// Mitsubishi GX Works2 project: OLD CRF BUFFER 22-01-223_F1   PLC: Q02/Q02H

PROGRAM MAIN
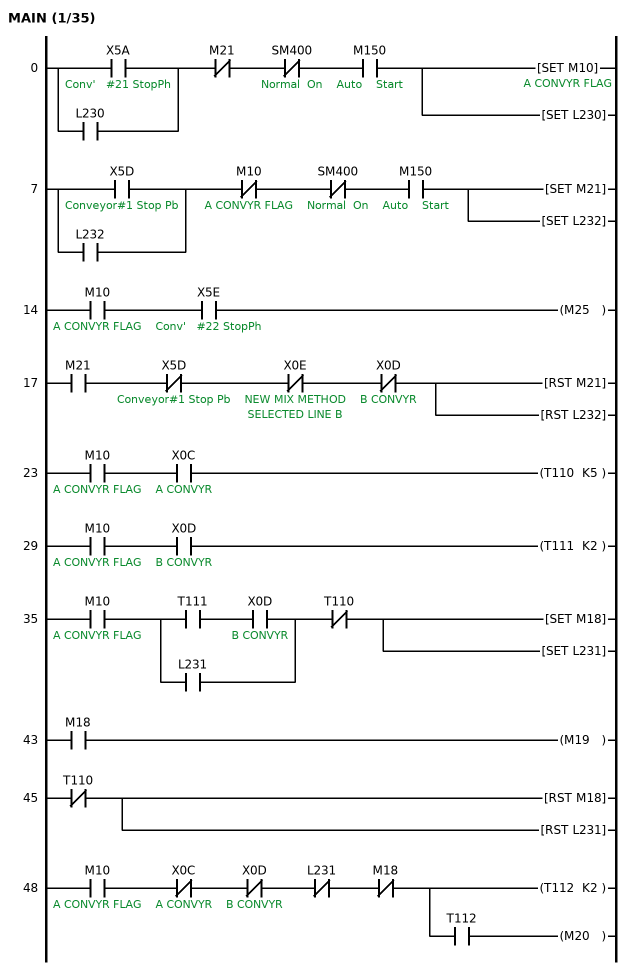
0     LD      X5A  ; Conv'   #21 StopPh
      OR      L230
      ANI     M21
      ANI     SM400  ; Normal  On
      AND     M150  ; Auto    Start
      SET     M10  ; A CONVYR FLAG
      SET     L230
7     LD      X5D  ; Conveyor#1 Stop Pb
      OR      L232
      ANI     M10  ; A CONVYR FLAG
      ANI     SM400  ; Normal  On
      AND     M150  ; Auto    Start
      SET     M21
      SET     L232
14    LD      M10  ; A CONVYR FLAG
      AND     X5E  ; Conv'   #22 StopPh
      OUT     M25
17    LD      M21
      ANI     X5D  ; Conveyor#1 Stop Pb
      ANI     X0E  ; NEW MIX METHOD  SELECTED LINE B
      ANI     X0D  ; B CONVYR
      RST     M21
      RST     L232
23    LD      M10  ; A CONVYR FLAG
      AND     X0C  ; A CONVYR
      OUT     T110 K5
29    LD      M10  ; A CONVYR FLAG
      AND     X0D  ; B CONVYR
      OUT     T111 K2
35    LD      M10  ; A CONVYR FLAG
      LD      T111
      AND     X0D  ; B CONVYR
      OR      L231
      ANB
      ANI     T110
      SET     M18
      SET     L231
43    LD      M18
      OUT     M19
45    LDI     T110
      RST     M18
      RST     L231
48    LD      M10  ; A CONVYR FLAG
      ANI     X0C  ; A CONVYR
      ANI     X0D  ; B CONVYR
      ANI     L231
      ANI     M18
      OUT     T112 K2
      AND     T112
      OUT     M20
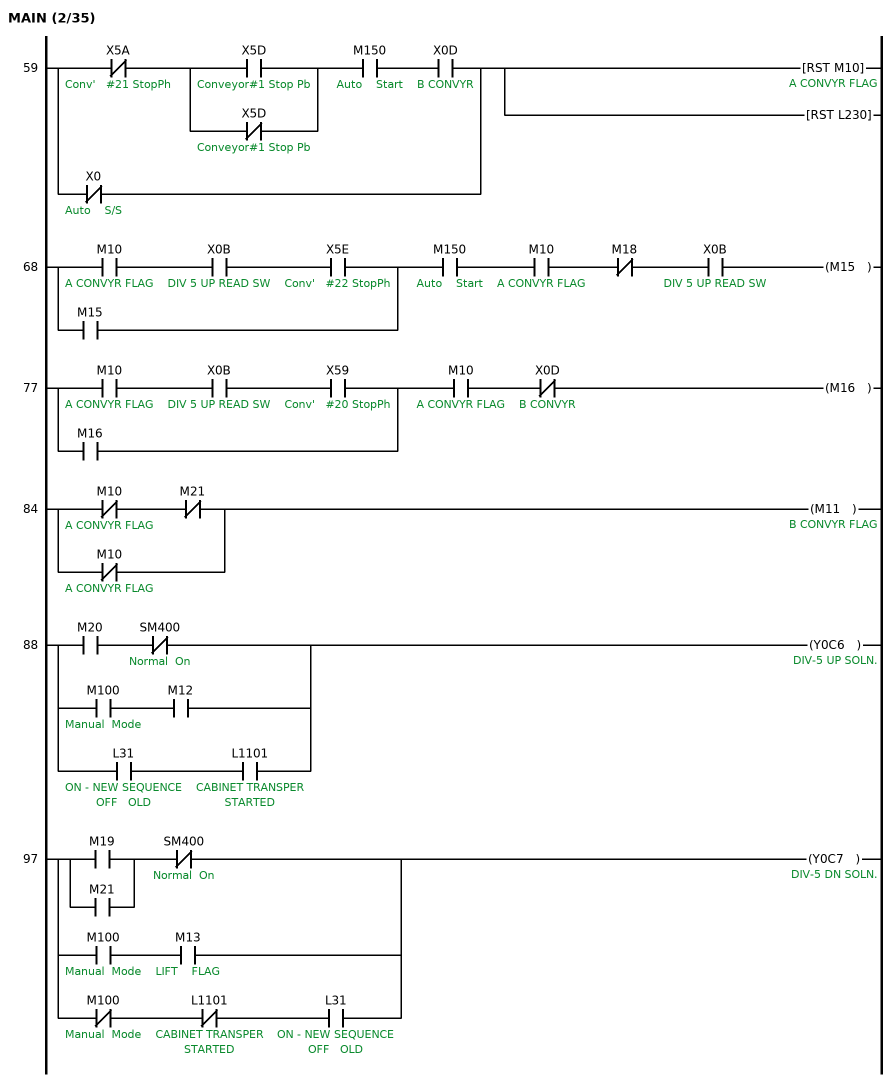
59    LDI     X5A  ; Conv'   #21 StopPh
      LD      X5D  ; Conveyor#1 Stop Pb
      ORI     X5D  ; Conveyor#1 Stop Pb
      ANB
      AND     M150  ; Auto    Start
      AND     X0D  ; B CONVYR
      ORI     X0  ; Auto    S/S
      RST     M10  ; A CONVYR FLAG
      RST     L230
68    LD      M10  ; A CONVYR FLAG
      AND     X0B  ; DIV 5 UP READ SW
      AND     X5E  ; Conv'   #22 StopPh
      OR      M15
      AND     M150  ; Auto    Start
      AND     M10  ; A CONVYR FLAG
      ANI     M18
      AND     X0B  ; DIV 5 UP READ SW
      OUT     M15
77    LD      M10  ; A CONVYR FLAG
      AND     X0B  ; DIV 5 UP READ SW
      AND     X59  ; Conv'   #20 StopPh
      OR      M16
      AND     M10  ; A CONVYR FLAG
      ANI     X0D  ; B CONVYR
      OUT     M16
84    LDI     M10  ; A CONVYR FLAG
      ANI     M21
      ORI     M10  ; A CONVYR FLAG
      OUT     M11  ; B CONVYR FLAG
88    LD      M20
      ANI     SM400  ; Normal  On
      LD      M100  ; Manual  Mode
      AND     M12
      ORB
      LD      L31  ; ON - NEW SEQUENCE OFF   OLD
      AND     L1101  ; CABINET TRANSPER STARTED
      ORB
      OUT     Y0C6  ; DIV-5 UP SOLN.
97    LD      M19
      OR      M21
      ANI     SM400  ; Normal  On
      LD      M100  ; Manual  Mode
      AND     M13  ; LIFT    FLAG
      ORB
      LDI     M100  ; Manual  Mode
      ANI     L1101  ; CABINET TRANSPER STARTED
      AND     L31  ; ON - NEW SEQUENCE OFF   OLD
      ORB
      OUT     Y0C7  ; DIV-5 DN SOLN.
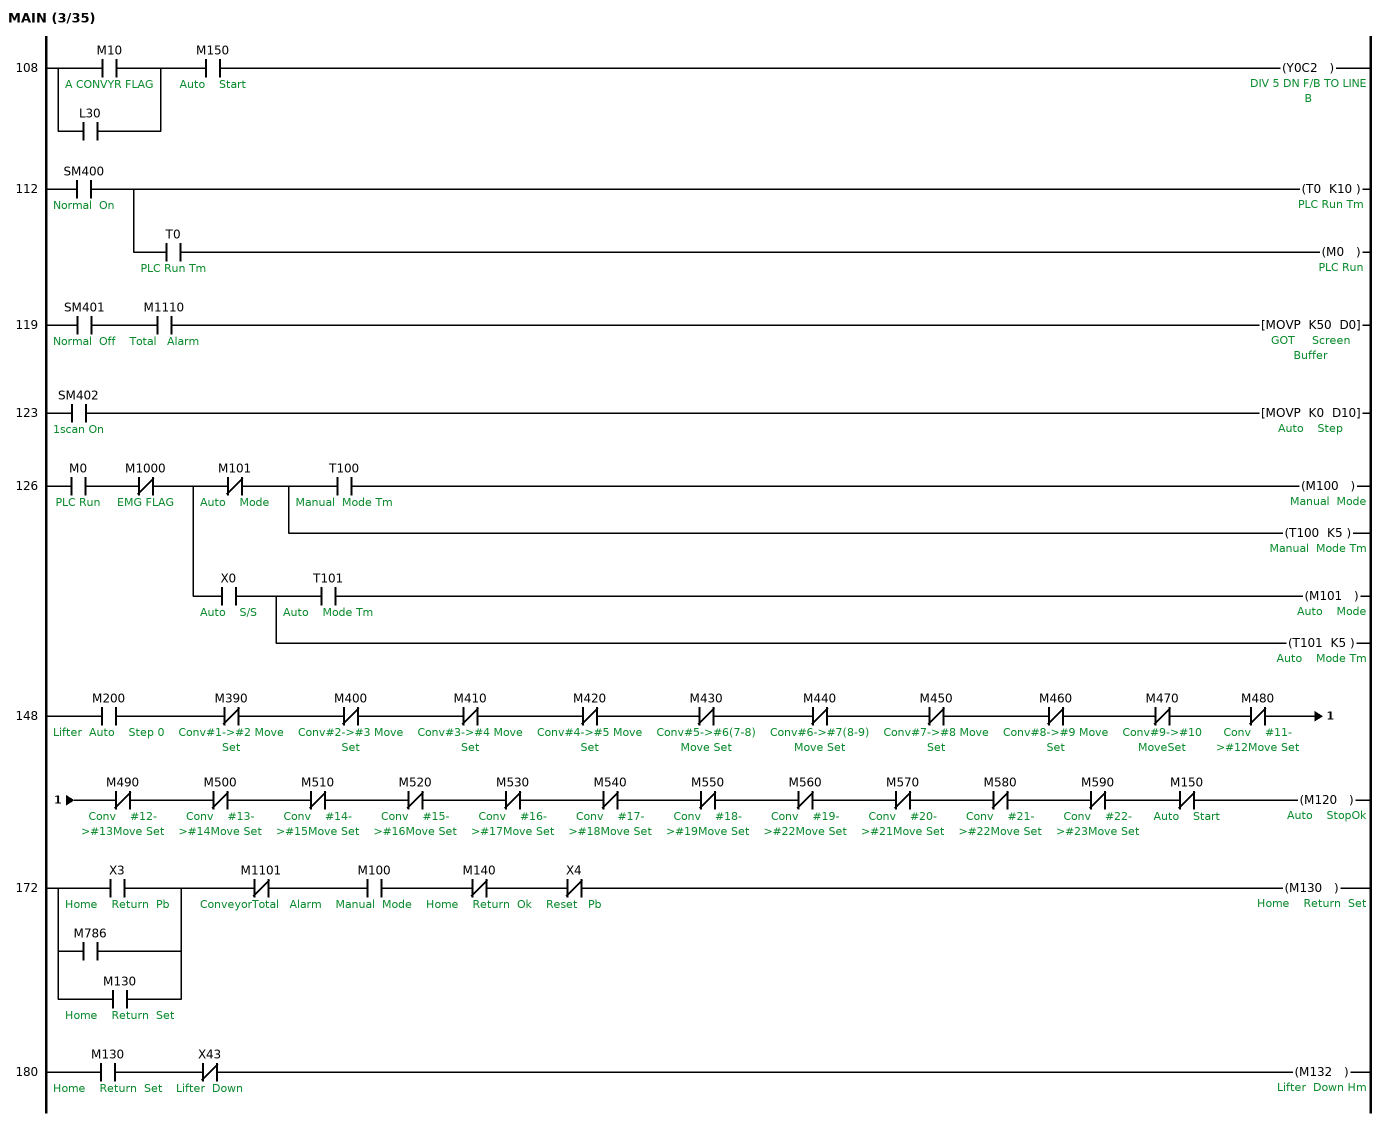
108   LD      M10  ; A CONVYR FLAG
      OR      L30
      AND     M150  ; Auto    Start
      OUT     Y0C2  ; DIV 5 DN F/B TO LINE B
112   LD      SM400  ; Normal  On
      OUT     T0 K10  ; PLC Run Tm
      AND     T0  ; PLC Run Tm
      OUT     M0  ; PLC Run
119   LD      SM401  ; Normal  Off
      AND     M1110  ; Total   Alarm
      MOVP    K50 D0  ; GOT     Screen  Buffer
123   LD      SM402  ; 1scan On
      MOVP    K0 D10  ; Auto    Step
126   LD      M0  ; PLC Run
      ANI     M1000  ; EMG FLAG
      MPS
      ANI     M101  ; Auto    Mode
      MPS
      AND     T100  ; Manual  Mode Tm
      OUT     M100  ; Manual  Mode
      MPP
      OUT     T100 K5  ; Manual  Mode Tm
      MPP
      AND     X0  ; Auto    S/S
      MPS
      AND     T101  ; Auto    Mode Tm
      OUT     M101  ; Auto    Mode
      MPP
      OUT     T101 K5  ; Auto    Mode Tm
148   LD      M200  ; Lifter  Auto    Step 0
      ANI     M390  ; Conv#1->#2 Move Set
      ANI     M400  ; Conv#2->#3 Move Set
      ANI     M410  ; Conv#3->#4 Move Set
      ANI     M420  ; Conv#4->#5 Move Set
      ANI     M430  ; Conv#5->#6(7-8) Move Set
      ANI     M440  ; Conv#6->#7(8-9) Move Set
      ANI     M450  ; Conv#7->#8 Move Set
      ANI     M460  ; Conv#8->#9 Move Set
      ANI     M470  ; Conv#9->#10 MoveSet
      ANI     M480  ; Conv    #11->#12Move Set
      ANI     M490  ; Conv    #12->#13Move Set
      ANI     M500  ; Conv    #13->#14Move Set
      ANI     M510  ; Conv    #14->#15Move Set
      ANI     M520  ; Conv    #15->#16Move Set
      ANI     M530  ; Conv    #16->#17Move Set
      ANI     M540  ; Conv    #17->#18Move Set
      ANI     M550  ; Conv    #18->#19Move Set
      ANI     M560  ; Conv    #19->#22Move Set
      ANI     M570  ; Conv    #20->#21Move Set
      ANI     M580  ; Conv    #21->#22Move Set
      ANI     M590  ; Conv    #22->#23Move Set
      ANI     M150  ; Auto    Start
      OUT     M120  ; Auto    StopOk
172   LD      X3  ; Home    Return  Pb
      OR      M786
      OR      M130  ; Home    Return  Set
      ANI     M1101  ; ConveyorTotal   Alarm
      AND     M100  ; Manual  Mode
      ANI     M140  ; Home    Return  Ok
      ANI     X4  ; Reset   Pb
      OUT     M130  ; Home    Return  Set
180   LD      M130  ; Home    Return  Set
      ANI     X43  ; Lifter  Down
      OUT     M132  ; Lifter  Down Hm
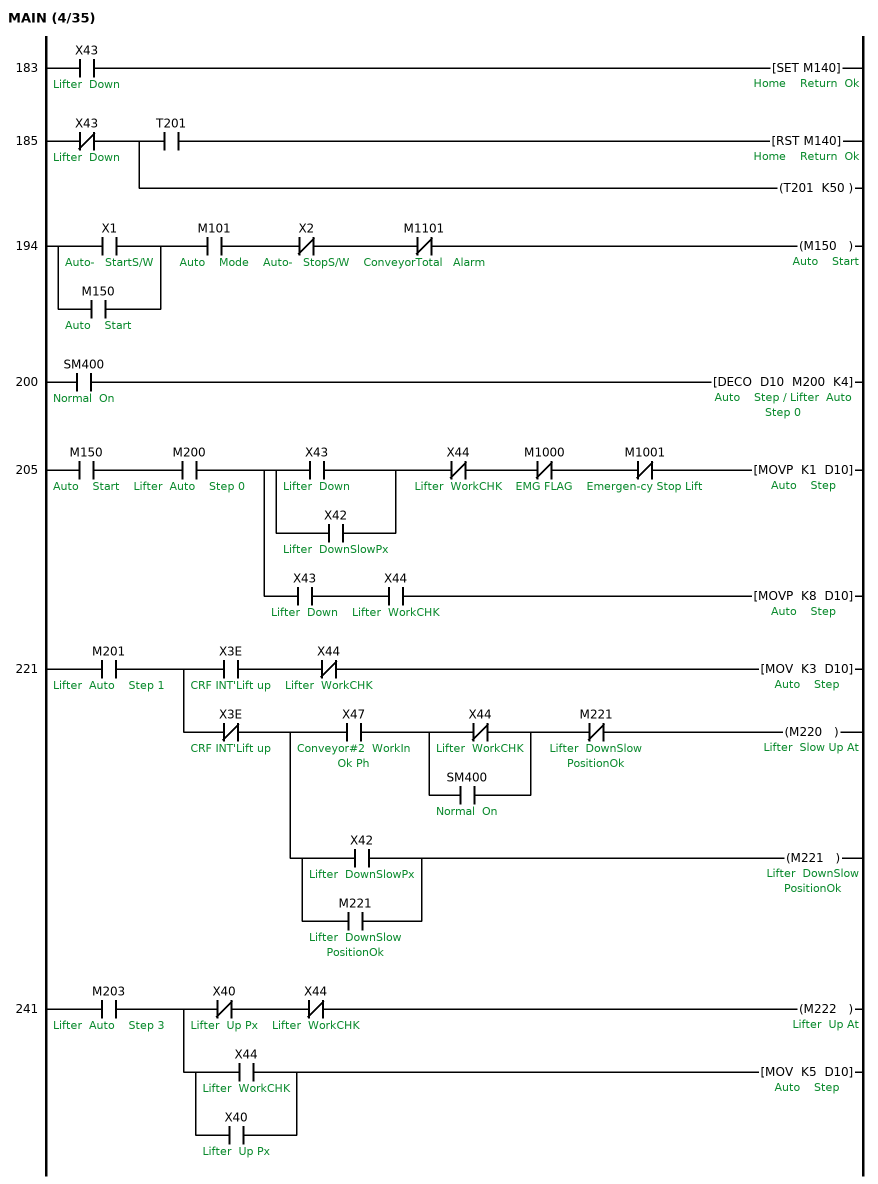
183   LD      X43  ; Lifter  Down
      SET     M140  ; Home    Return  Ok
185   LDI     X43  ; Lifter  Down
      MPS
      AND     T201
      RST     M140  ; Home    Return  Ok
      MPP
      OUT     T201 K50
194   LD      X1  ; Auto-   StartS/W
      OR      M150  ; Auto    Start
      AND     M101  ; Auto    Mode
      ANI     X2  ; Auto-   StopS/W
      ANI     M1101  ; ConveyorTotal   Alarm
      OUT     M150  ; Auto    Start
200   LD      SM400  ; Normal  On
      DECO    D10 M200 K4
205   LD      M150  ; Auto    Start
      AND     M200  ; Lifter  Auto    Step 0
      MPS
      LD      X43  ; Lifter  Down
      OR      X42  ; Lifter  DownSlowPx
      ANB
      ANI     X44  ; Lifter  WorkCHK
      ANI     M1000  ; EMG FLAG
      ANI     M1001  ; Emergen-cy Stop Lift
      MOVP    K1 D10
      MPP
      AND     X43  ; Lifter  Down
      AND     X44  ; Lifter  WorkCHK
      MOVP    K8 D10
221   LD      M201  ; Lifter  Auto    Step 1
      MPS
      AND     X3E  ; CRF INT'Lift up
      ANI     X44  ; Lifter  WorkCHK
      MOV     K3 D10
      MPP
      ANI     X3E  ; CRF INT'Lift up
      MPS
      AND     X47  ; Conveyor#2  WorkIn Ok Ph
      LDI     X44  ; Lifter  WorkCHK
      OR      SM400  ; Normal  On
      ANB
      ANI     M221  ; Lifter  DownSlowPositionOk
      OUT     M220  ; Lifter  Slow Up At
      MPP
      LD      X42  ; Lifter  DownSlowPx
      OR      M221  ; Lifter  DownSlowPositionOk
      ANB
      OUT     M221  ; Lifter  DownSlowPositionOk
241   LD      M203  ; Lifter  Auto    Step 3
      MPS
      ANI     X40  ; Lifter  Up Px
      ANI     X44  ; Lifter  WorkCHK
      OUT     M222  ; Lifter  Up At
      MPP
      LD      X44  ; Lifter  WorkCHK
      OR      X40  ; Lifter  Up Px
      ANB
      MOV     K5 D10
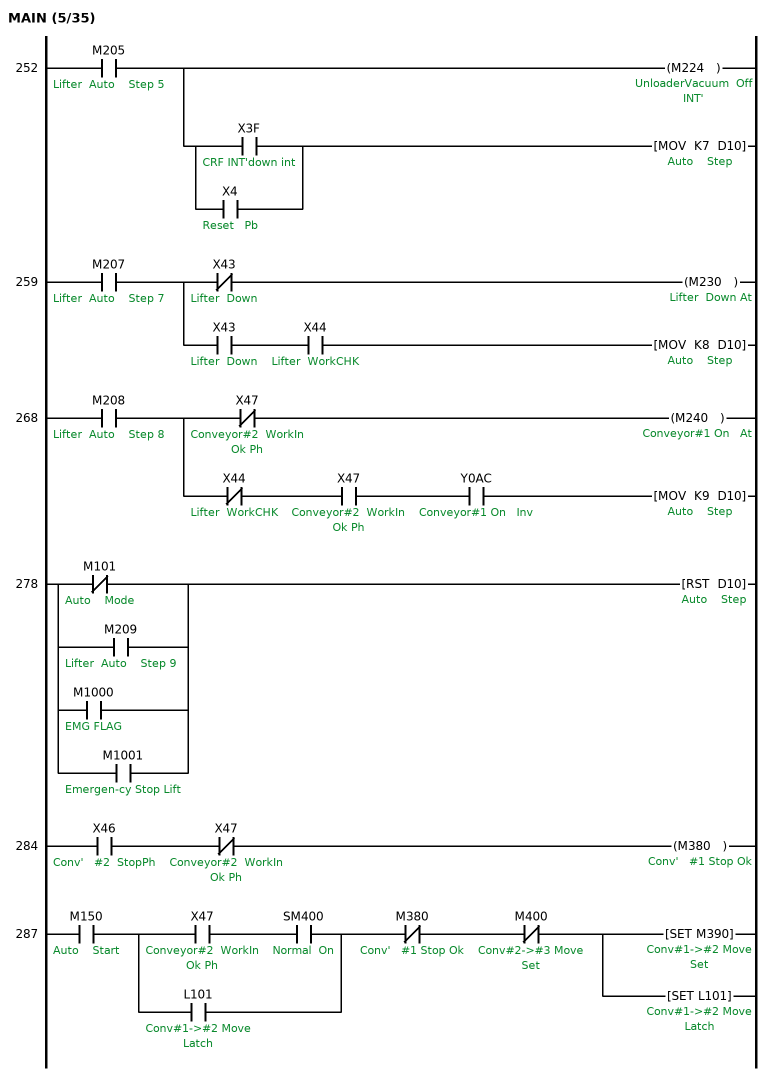
252   LD      M205  ; Lifter  Auto    Step 5
      OUT     M224  ; UnloaderVacuum  Off INT'
      LD      X3F  ; CRF INT'down int
      OR      X4  ; Reset   Pb
      ANB
      MOV     K7 D10
259   LD      M207  ; Lifter  Auto    Step 7
      MPS
      ANI     X43  ; Lifter  Down
      OUT     M230  ; Lifter  Down At
      MPP
      AND     X43  ; Lifter  Down
      AND     X44  ; Lifter  WorkCHK
      MOV     K8 D10
268   LD      M208  ; Lifter  Auto    Step 8
      MPS
      ANI     X47  ; Conveyor#2  WorkIn Ok Ph
      OUT     M240  ; Conveyor#1 On   At
      MPP
      ANI     X44  ; Lifter  WorkCHK
      AND     X47  ; Conveyor#2  WorkIn Ok Ph
      AND     Y0AC  ; Conveyor#1 On   Inv
      MOV     K9 D10
278   LDI     M101  ; Auto    Mode
      OR      M209  ; Lifter  Auto    Step 9
      OR      M1000  ; EMG FLAG
      OR      M1001  ; Emergen-cy Stop Lift
      RST     D10  ; Auto    Step
284   LD      X46  ; Conv'   #2  StopPh
      ANI     X47  ; Conveyor#2  WorkIn Ok Ph
      OUT     M380  ; Conv'   #1 Stop Ok
287   LD      M150  ; Auto    Start
      LD      X47  ; Conveyor#2  WorkIn Ok Ph
      AND     SM400  ; Normal  On
      OR      L101  ; Conv#1->#2 Move Latch
      ANB
      ANI     M380  ; Conv'   #1 Stop Ok
      ANI     M400  ; Conv#2->#3 Move Set
      SET     M390  ; Conv#1->#2 Move Set
      SET     L101  ; Conv#1->#2 Move Latch
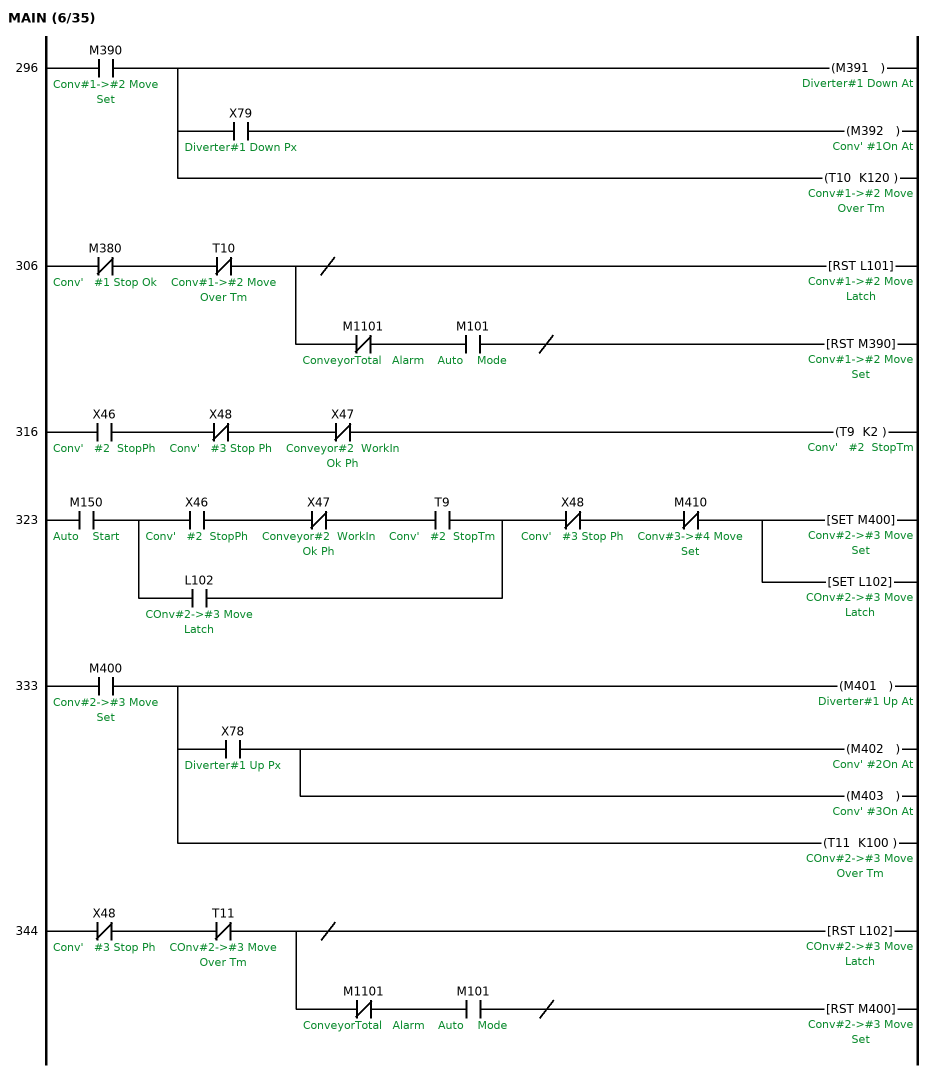
296   LD      M390  ; Conv#1->#2 Move Set
      OUT     M391  ; Diverter#1 Down At
      MPS
      AND     X79  ; Diverter#1 Down Px
      OUT     M392  ; Conv' #1On At
      MPP
      OUT     T10 K120  ; Conv#1->#2 Move Over Tm
306   LDI     M380  ; Conv'   #1 Stop Ok
      ANI     T10  ; Conv#1->#2 Move Over Tm
      MPS
      INV
      RST     L101  ; Conv#1->#2 Move Latch
      MPP
      ANI     M1101  ; ConveyorTotal   Alarm
      AND     M101  ; Auto    Mode
      INV
      RST     M390  ; Conv#1->#2 Move Set
316   LD      X46  ; Conv'   #2  StopPh
      ANI     X48  ; Conv'   #3 Stop Ph
      ANI     X47  ; Conveyor#2  WorkIn Ok Ph
      OUT     T9 K2  ; Conv'   #2  StopTm
323   LD      M150  ; Auto    Start
      LD      X46  ; Conv'   #2  StopPh
      ANI     X47  ; Conveyor#2  WorkIn Ok Ph
      AND     T9  ; Conv'   #2  StopTm
      OR      L102  ; COnv#2->#3 Move Latch
      ANB
      ANI     X48  ; Conv'   #3 Stop Ph
      ANI     M410  ; Conv#3->#4 Move Set
      SET     M400  ; Conv#2->#3 Move Set
      SET     L102  ; COnv#2->#3 Move Latch
333   LD      M400  ; Conv#2->#3 Move Set
      OUT     M401  ; Diverter#1 Up At
      MPS
      AND     X78  ; Diverter#1 Up Px
      OUT     M402  ; Conv' #2On At
      OUT     M403  ; Conv' #3On At
      MPP
      OUT     T11 K100  ; COnv#2->#3 Move Over Tm
344   LDI     X48  ; Conv'   #3 Stop Ph
      ANI     T11  ; COnv#2->#3 Move Over Tm
      MPS
      INV
      RST     L102  ; COnv#2->#3 Move Latch
      MPP
      ANI     M1101  ; ConveyorTotal   Alarm
      AND     M101  ; Auto    Mode
      INV
      RST     M400  ; Conv#2->#3 Move Set
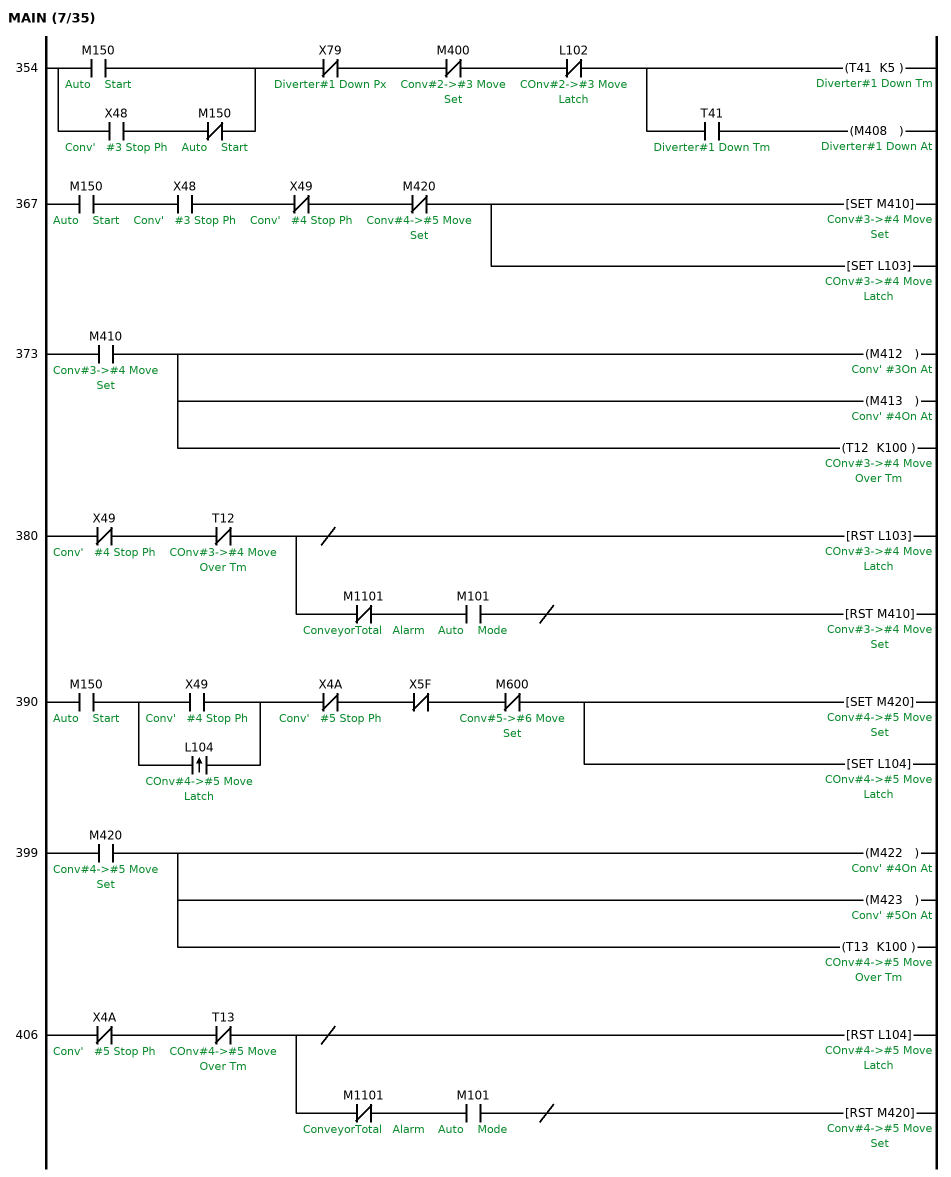
354   LD      M150  ; Auto    Start
      LD      X48  ; Conv'   #3 Stop Ph
      ANI     M150  ; Auto    Start
      ORB
      ANI     X79  ; Diverter#1 Down Px
      ANI     M400  ; Conv#2->#3 Move Set
      ANI     L102  ; COnv#2->#3 Move Latch
      OUT     T41 K5  ; Diverter#1 Down Tm
      AND     T41  ; Diverter#1 Down Tm
      OUT     M408  ; Diverter#1 Down At
367   LD      M150  ; Auto    Start
      AND     X48  ; Conv'   #3 Stop Ph
      ANI     X49  ; Conv'   #4 Stop Ph
      ANI     M420  ; Conv#4->#5 Move Set
      SET     M410  ; Conv#3->#4 Move Set
      SET     L103  ; COnv#3->#4 Move Latch
373   LD      M410  ; Conv#3->#4 Move Set
      OUT     M412  ; Conv' #3On At
      OUT     M413  ; Conv' #4On At
      OUT     T12 K100  ; COnv#3->#4 Move Over Tm
380   LDI     X49  ; Conv'   #4 Stop Ph
      ANI     T12  ; COnv#3->#4 Move Over Tm
      MPS
      INV
      RST     L103  ; COnv#3->#4 Move Latch
      MPP
      ANI     M1101  ; ConveyorTotal   Alarm
      AND     M101  ; Auto    Mode
      INV
      RST     M410  ; Conv#3->#4 Move Set
390   LD      M150  ; Auto    Start
      LD      X49  ; Conv'   #4 Stop Ph
      ORP     L104  ; COnv#4->#5 Move Latch
      ANB
      ANI     X4A  ; Conv'   #5 Stop Ph
      ANI     X5F
      ANI     M600  ; Conv#5->#6 Move Set
      SET     M420  ; Conv#4->#5 Move Set
      SET     L104  ; COnv#4->#5 Move Latch
399   LD      M420  ; Conv#4->#5 Move Set
      OUT     M422  ; Conv' #4On At
      OUT     M423  ; Conv' #5On At
      OUT     T13 K100  ; COnv#4->#5 Move Over Tm
406   LDI     X4A  ; Conv'   #5 Stop Ph
      ANI     T13  ; COnv#4->#5 Move Over Tm
      MPS
      INV
      RST     L104  ; COnv#4->#5 Move Latch
      MPP
      ANI     M1101  ; ConveyorTotal   Alarm
      AND     M101  ; Auto    Mode
      INV
      RST     M420  ; Conv#4->#5 Move Set
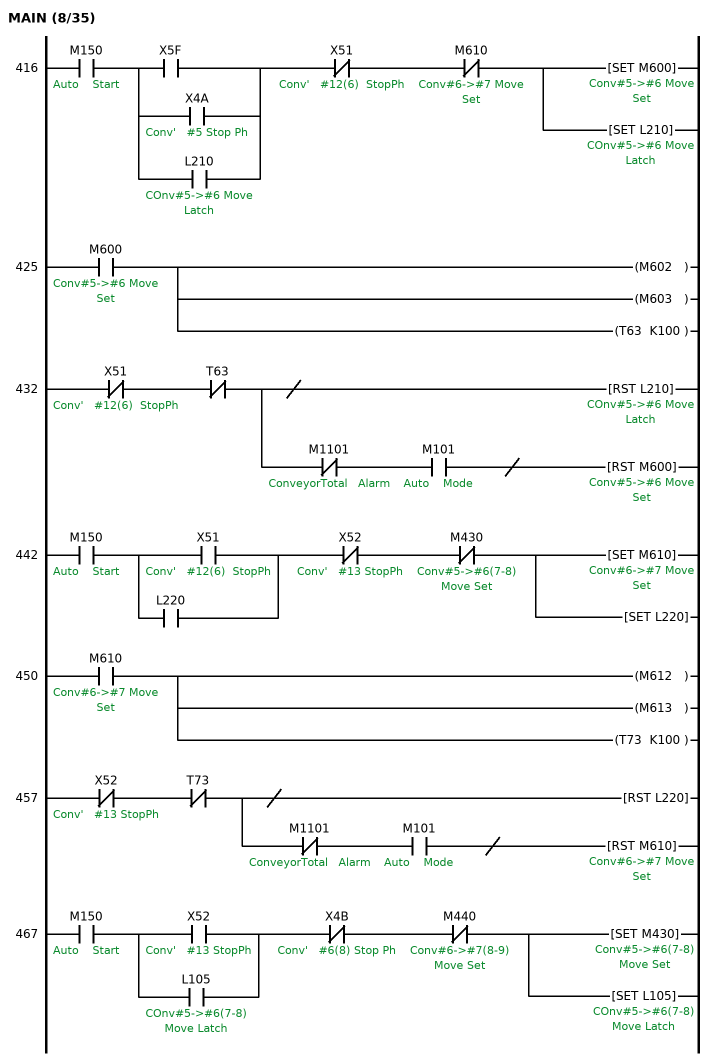
416   LD      M150  ; Auto    Start
      LD      X5F
      OR      X4A  ; Conv'   #5 Stop Ph
      OR      L210  ; COnv#5->#6 Move Latch
      ANB
      ANI     X51  ; Conv'   #12(6)  StopPh
      ANI     M610  ; Conv#6->#7 Move Set
      SET     M600  ; Conv#5->#6 Move Set
      SET     L210  ; COnv#5->#6 Move Latch
425   LD      M600  ; Conv#5->#6 Move Set
      OUT     M602
      OUT     M603
      OUT     T63 K100
432   LDI     X51  ; Conv'   #12(6)  StopPh
      ANI     T63
      MPS
      INV
      RST     L210  ; COnv#5->#6 Move Latch
      MPP
      ANI     M1101  ; ConveyorTotal   Alarm
      AND     M101  ; Auto    Mode
      INV
      RST     M600  ; Conv#5->#6 Move Set
442   LD      M150  ; Auto    Start
      LD      X51  ; Conv'   #12(6)  StopPh
      OR      L220
      ANB
      ANI     X52  ; Conv'   #13 StopPh
      ANI     M430  ; Conv#5->#6(7-8) Move Set
      SET     M610  ; Conv#6->#7 Move Set
      SET     L220
450   LD      M610  ; Conv#6->#7 Move Set
      OUT     M612
      OUT     M613
      OUT     T73 K100
457   LDI     X52  ; Conv'   #13 StopPh
      ANI     T73
      MPS
      INV
      RST     L220
      MPP
      ANI     M1101  ; ConveyorTotal   Alarm
      AND     M101  ; Auto    Mode
      INV
      RST     M610  ; Conv#6->#7 Move Set
467   LD      M150  ; Auto    Start
      LD      X52  ; Conv'   #13 StopPh
      OR      L105  ; COnv#5->#6(7-8) Move Latch
      ANB
      ANI     X4B  ; Conv'   #6(8) Stop Ph
      ANI     M440  ; Conv#6->#7(8-9) Move Set
      SET     M430  ; Conv#5->#6(7-8) Move Set
      SET     L105  ; COnv#5->#6(7-8) Move Latch
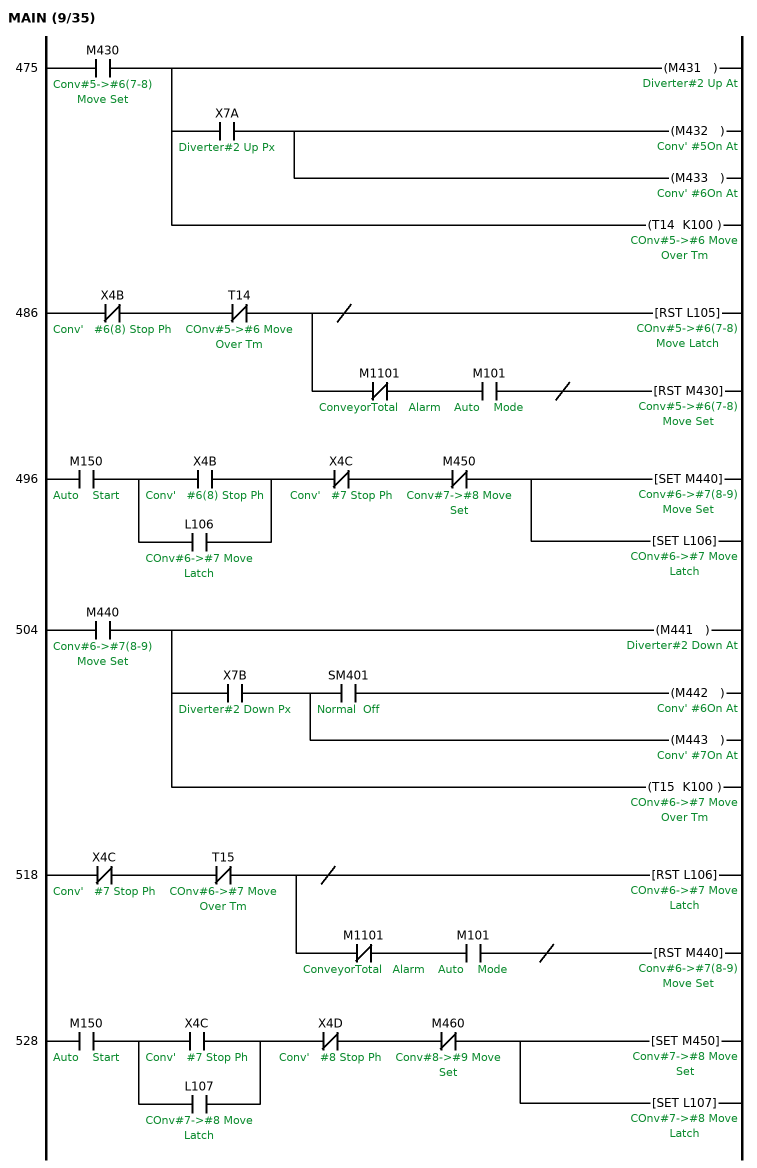
475   LD      M430  ; Conv#5->#6(7-8) Move Set
      OUT     M431  ; Diverter#2 Up At
      MPS
      AND     X7A  ; Diverter#2 Up Px
      OUT     M432  ; Conv' #5On At
      OUT     M433  ; Conv' #6On At
      MPP
      OUT     T14 K100  ; COnv#5->#6 Move Over Tm
486   LDI     X4B  ; Conv'   #6(8) Stop Ph
      ANI     T14  ; COnv#5->#6 Move Over Tm
      MPS
      INV
      RST     L105  ; COnv#5->#6(7-8) Move Latch
      MPP
      ANI     M1101  ; ConveyorTotal   Alarm
      AND     M101  ; Auto    Mode
      INV
      RST     M430  ; Conv#5->#6(7-8) Move Set
496   LD      M150  ; Auto    Start
      LD      X4B  ; Conv'   #6(8) Stop Ph
      OR      L106  ; COnv#6->#7 Move Latch
      ANB
      ANI     X4C  ; Conv'   #7 Stop Ph
      ANI     M450  ; Conv#7->#8 Move Set
      SET     M440  ; Conv#6->#7(8-9) Move Set
      SET     L106  ; COnv#6->#7 Move Latch
504   LD      M440  ; Conv#6->#7(8-9) Move Set
      OUT     M441  ; Diverter#2 Down At
      MPS
      AND     X7B  ; Diverter#2 Down Px
      MPS
      AND     SM401  ; Normal  Off
      OUT     M442  ; Conv' #6On At
      MPP
      OUT     M443  ; Conv' #7On At
      MPP
      OUT     T15 K100  ; COnv#6->#7 Move Over Tm
518   LDI     X4C  ; Conv'   #7 Stop Ph
      ANI     T15  ; COnv#6->#7 Move Over Tm
      MPS
      INV
      RST     L106  ; COnv#6->#7 Move Latch
      MPP
      ANI     M1101  ; ConveyorTotal   Alarm
      AND     M101  ; Auto    Mode
      INV
      RST     M440  ; Conv#6->#7(8-9) Move Set
528   LD      M150  ; Auto    Start
      LD      X4C  ; Conv'   #7 Stop Ph
      OR      L107  ; COnv#7->#8 Move Latch
      ANB
      ANI     X4D  ; Conv'   #8 Stop Ph
      ANI     M460  ; Conv#8->#9 Move Set
      SET     M450  ; Conv#7->#8 Move Set
      SET     L107  ; COnv#7->#8 Move Latch
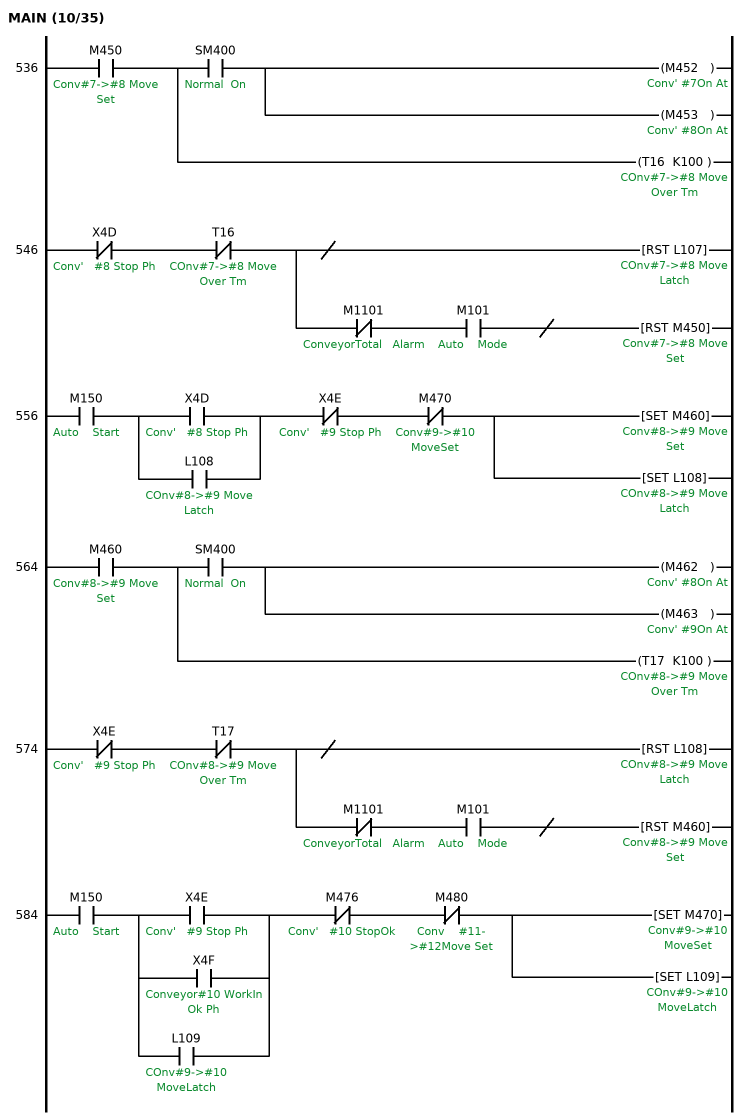
536   LD      M450  ; Conv#7->#8 Move Set
      MPS
      AND     SM400  ; Normal  On
      OUT     M452  ; Conv' #7On At
      OUT     M453  ; Conv' #8On At
      MPP
      OUT     T16 K100  ; COnv#7->#8 Move Over Tm
546   LDI     X4D  ; Conv'   #8 Stop Ph
      ANI     T16  ; COnv#7->#8 Move Over Tm
      MPS
      INV
      RST     L107  ; COnv#7->#8 Move Latch
      MPP
      ANI     M1101  ; ConveyorTotal   Alarm
      AND     M101  ; Auto    Mode
      INV
      RST     M450  ; Conv#7->#8 Move Set
556   LD      M150  ; Auto    Start
      LD      X4D  ; Conv'   #8 Stop Ph
      OR      L108  ; COnv#8->#9 Move Latch
      ANB
      ANI     X4E  ; Conv'   #9 Stop Ph
      ANI     M470  ; Conv#9->#10 MoveSet
      SET     M460  ; Conv#8->#9 Move Set
      SET     L108  ; COnv#8->#9 Move Latch
564   LD      M460  ; Conv#8->#9 Move Set
      MPS
      AND     SM400  ; Normal  On
      OUT     M462  ; Conv' #8On At
      OUT     M463  ; Conv' #9On At
      MPP
      OUT     T17 K100  ; COnv#8->#9 Move Over Tm
574   LDI     X4E  ; Conv'   #9 Stop Ph
      ANI     T17  ; COnv#8->#9 Move Over Tm
      MPS
      INV
      RST     L108  ; COnv#8->#9 Move Latch
      MPP
      ANI     M1101  ; ConveyorTotal   Alarm
      AND     M101  ; Auto    Mode
      INV
      RST     M460  ; Conv#8->#9 Move Set
584   LD      M150  ; Auto    Start
      LD      X4E  ; Conv'   #9 Stop Ph
      OR      X4F  ; Conveyor#10 WorkIn Ok Ph
      OR      L109  ; COnv#9->#10 MoveLatch
      ANB
      ANI     M476  ; Conv'   #10 StopOk
      ANI     M480  ; Conv    #11->#12Move Set
      SET     M470  ; Conv#9->#10 MoveSet
      SET     L109  ; COnv#9->#10 MoveLatch
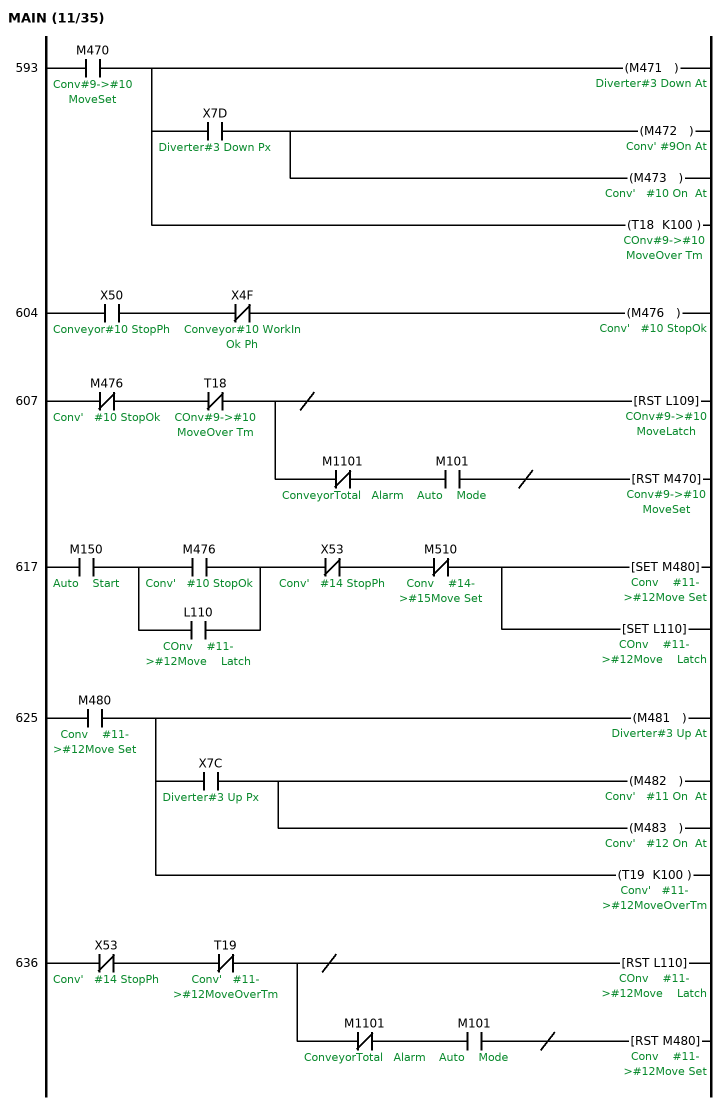
593   LD      M470  ; Conv#9->#10 MoveSet
      OUT     M471  ; Diverter#3 Down At
      MPS
      AND     X7D  ; Diverter#3 Down Px
      OUT     M472  ; Conv' #9On At
      OUT     M473  ; Conv'   #10 On  At
      MPP
      OUT     T18 K100  ; COnv#9->#10 MoveOver Tm
604   LD      X50  ; Conveyor#10 StopPh
      ANI     X4F  ; Conveyor#10 WorkIn Ok Ph
      OUT     M476  ; Conv'   #10 StopOk
607   LDI     M476  ; Conv'   #10 StopOk
      ANI     T18  ; COnv#9->#10 MoveOver Tm
      MPS
      INV
      RST     L109  ; COnv#9->#10 MoveLatch
      MPP
      ANI     M1101  ; ConveyorTotal   Alarm
      AND     M101  ; Auto    Mode
      INV
      RST     M470  ; Conv#9->#10 MoveSet
617   LD      M150  ; Auto    Start
      LD      M476  ; Conv'   #10 StopOk
      OR      L110  ; COnv    #11->#12Move    Latch
      ANB
      ANI     X53  ; Conv'   #14 StopPh
      ANI     M510  ; Conv    #14->#15Move Set
      SET     M480  ; Conv    #11->#12Move Set
      SET     L110  ; COnv    #11->#12Move    Latch
625   LD      M480  ; Conv    #11->#12Move Set
      OUT     M481  ; Diverter#3 Up At
      MPS
      AND     X7C  ; Diverter#3 Up Px
      OUT     M482  ; Conv'   #11 On  At
      OUT     M483  ; Conv'   #12 On  At
      MPP
      OUT     T19 K100  ; Conv'   #11->#12MoveOverTm
636   LDI     X53  ; Conv'   #14 StopPh
      ANI     T19  ; Conv'   #11->#12MoveOverTm
      MPS
      INV
      RST     L110  ; COnv    #11->#12Move    Latch
      MPP
      ANI     M1101  ; ConveyorTotal   Alarm
      AND     M101  ; Auto    Mode
      INV
      RST     M480  ; Conv    #11->#12Move Set
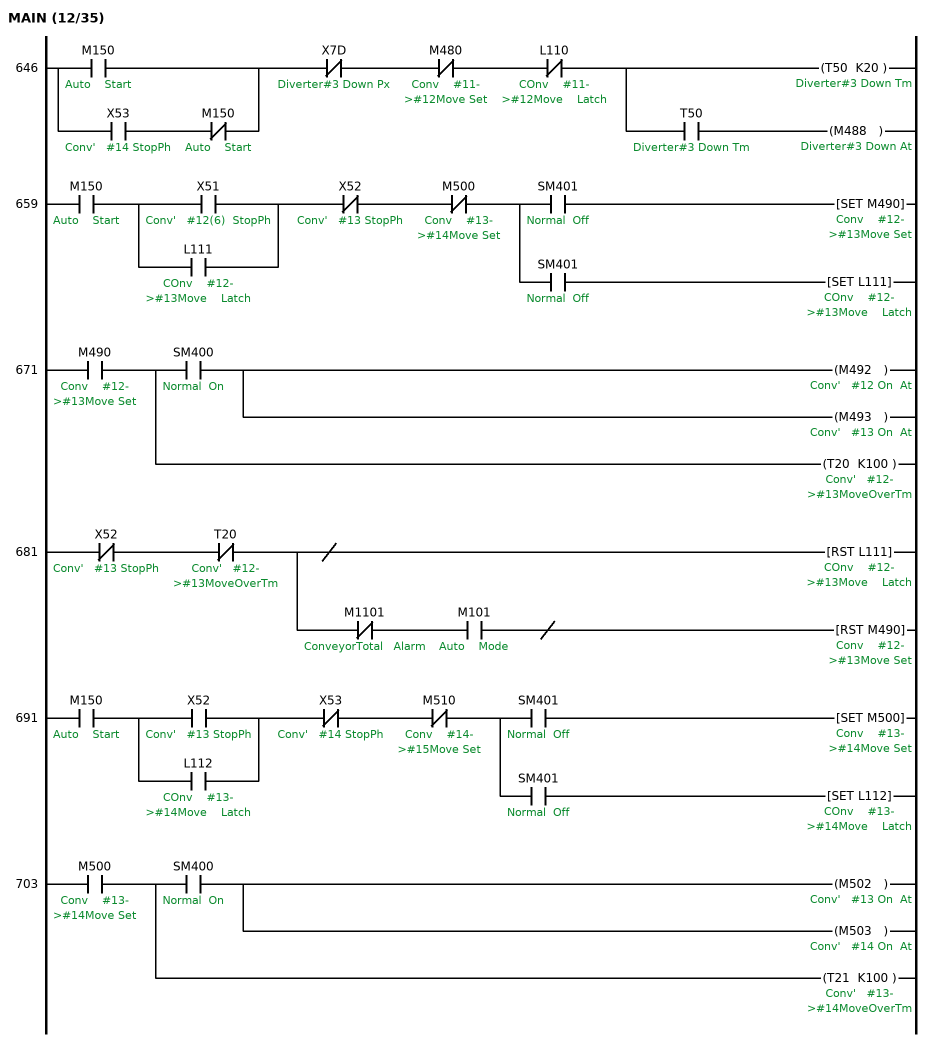
646   LD      M150  ; Auto    Start
      LD      X53  ; Conv'   #14 StopPh
      ANI     M150  ; Auto    Start
      ORB
      ANI     X7D  ; Diverter#3 Down Px
      ANI     M480  ; Conv    #11->#12Move Set
      ANI     L110  ; COnv    #11->#12Move    Latch
      OUT     T50 K20  ; Diverter#3 Down Tm
      AND     T50  ; Diverter#3 Down Tm
      OUT     M488  ; Diverter#3 Down At
659   LD      M150  ; Auto    Start
      LD      X51  ; Conv'   #12(6)  StopPh
      OR      L111  ; COnv    #12->#13Move    Latch
      ANB
      ANI     X52  ; Conv'   #13 StopPh
      ANI     M500  ; Conv    #13->#14Move Set
      MPS
      AND     SM401  ; Normal  Off
      SET     M490  ; Conv    #12->#13Move Set
      MPP
      AND     SM401  ; Normal  Off
      SET     L111  ; COnv    #12->#13Move    Latch
671   LD      M490  ; Conv    #12->#13Move Set
      MPS
      AND     SM400  ; Normal  On
      OUT     M492  ; Conv'   #12 On  At
      OUT     M493  ; Conv'   #13 On  At
      MPP
      OUT     T20 K100  ; Conv'   #12->#13MoveOverTm
681   LDI     X52  ; Conv'   #13 StopPh
      ANI     T20  ; Conv'   #12->#13MoveOverTm
      MPS
      INV
      RST     L111  ; COnv    #12->#13Move    Latch
      MPP
      ANI     M1101  ; ConveyorTotal   Alarm
      AND     M101  ; Auto    Mode
      INV
      RST     M490  ; Conv    #12->#13Move Set
691   LD      M150  ; Auto    Start
      LD      X52  ; Conv'   #13 StopPh
      OR      L112  ; COnv    #13->#14Move    Latch
      ANB
      ANI     X53  ; Conv'   #14 StopPh
      ANI     M510  ; Conv    #14->#15Move Set
      MPS
      AND     SM401  ; Normal  Off
      SET     M500  ; Conv    #13->#14Move Set
      MPP
      AND     SM401  ; Normal  Off
      SET     L112  ; COnv    #13->#14Move    Latch
703   LD      M500  ; Conv    #13->#14Move Set
      MPS
      AND     SM400  ; Normal  On
      OUT     M502  ; Conv'   #13 On  At
      OUT     M503  ; Conv'   #14 On  At
      MPP
      OUT     T21 K100  ; Conv'   #13->#14MoveOverTm
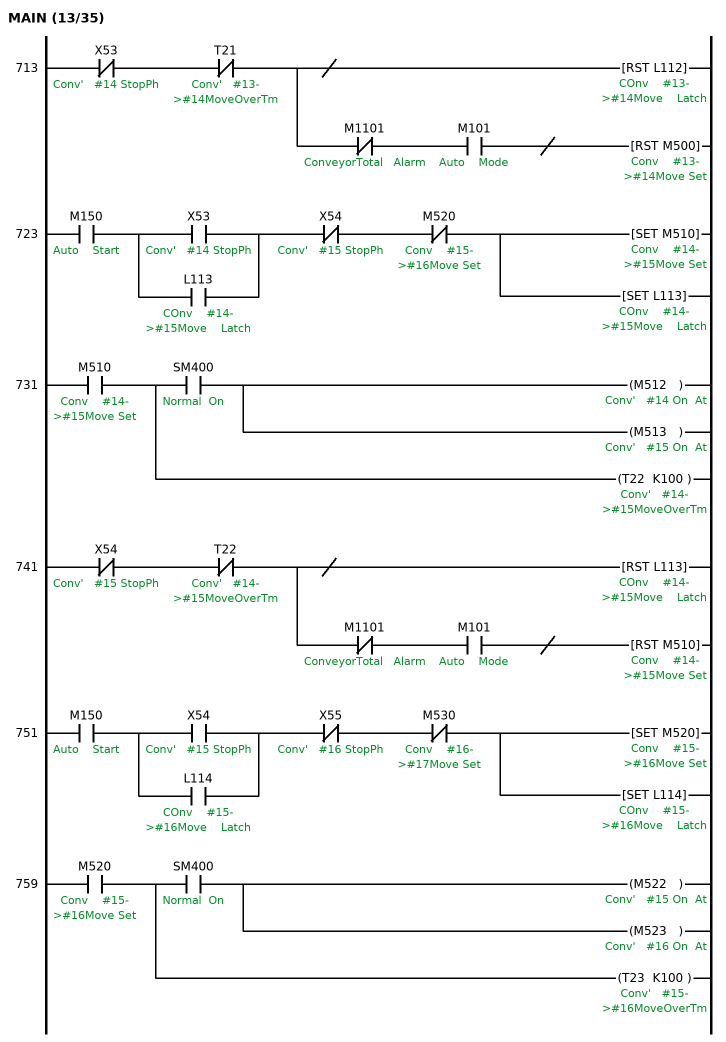
713   LDI     X53  ; Conv'   #14 StopPh
      ANI     T21  ; Conv'   #13->#14MoveOverTm
      MPS
      INV
      RST     L112  ; COnv    #13->#14Move    Latch
      MPP
      ANI     M1101  ; ConveyorTotal   Alarm
      AND     M101  ; Auto    Mode
      INV
      RST     M500  ; Conv    #13->#14Move Set
723   LD      M150  ; Auto    Start
      LD      X53  ; Conv'   #14 StopPh
      OR      L113  ; COnv    #14->#15Move    Latch
      ANB
      ANI     X54  ; Conv'   #15 StopPh
      ANI     M520  ; Conv    #15->#16Move Set
      SET     M510  ; Conv    #14->#15Move Set
      SET     L113  ; COnv    #14->#15Move    Latch
731   LD      M510  ; Conv    #14->#15Move Set
      MPS
      AND     SM400  ; Normal  On
      OUT     M512  ; Conv'   #14 On  At
      OUT     M513  ; Conv'   #15 On  At
      MPP
      OUT     T22 K100  ; Conv'   #14->#15MoveOverTm
741   LDI     X54  ; Conv'   #15 StopPh
      ANI     T22  ; Conv'   #14->#15MoveOverTm
      MPS
      INV
      RST     L113  ; COnv    #14->#15Move    Latch
      MPP
      ANI     M1101  ; ConveyorTotal   Alarm
      AND     M101  ; Auto    Mode
      INV
      RST     M510  ; Conv    #14->#15Move Set
751   LD      M150  ; Auto    Start
      LD      X54  ; Conv'   #15 StopPh
      OR      L114  ; COnv    #15->#16Move    Latch
      ANB
      ANI     X55  ; Conv'   #16 StopPh
      ANI     M530  ; Conv    #16->#17Move Set
      SET     M520  ; Conv    #15->#16Move Set
      SET     L114  ; COnv    #15->#16Move    Latch
759   LD      M520  ; Conv    #15->#16Move Set
      MPS
      AND     SM400  ; Normal  On
      OUT     M522  ; Conv'   #15 On  At
      OUT     M523  ; Conv'   #16 On  At
      MPP
      OUT     T23 K100  ; Conv'   #15->#16MoveOverTm
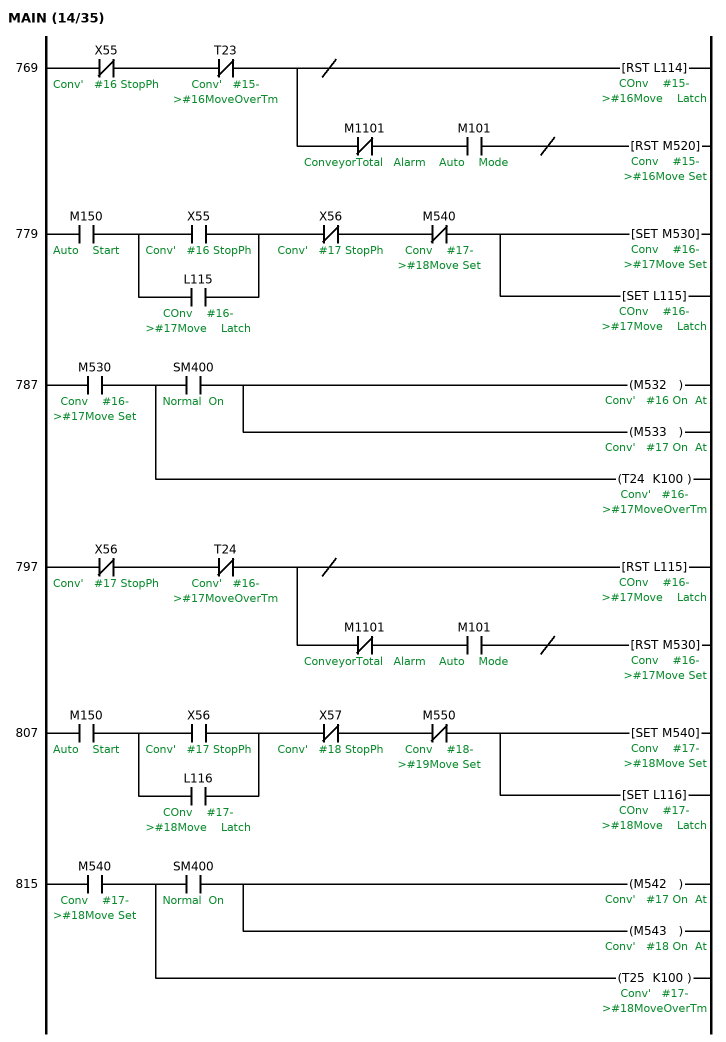
769   LDI     X55  ; Conv'   #16 StopPh
      ANI     T23  ; Conv'   #15->#16MoveOverTm
      MPS
      INV
      RST     L114  ; COnv    #15->#16Move    Latch
      MPP
      ANI     M1101  ; ConveyorTotal   Alarm
      AND     M101  ; Auto    Mode
      INV
      RST     M520  ; Conv    #15->#16Move Set
779   LD      M150  ; Auto    Start
      LD      X55  ; Conv'   #16 StopPh
      OR      L115  ; COnv    #16->#17Move    Latch
      ANB
      ANI     X56  ; Conv'   #17 StopPh
      ANI     M540  ; Conv    #17->#18Move Set
      SET     M530  ; Conv    #16->#17Move Set
      SET     L115  ; COnv    #16->#17Move    Latch
787   LD      M530  ; Conv    #16->#17Move Set
      MPS
      AND     SM400  ; Normal  On
      OUT     M532  ; Conv'   #16 On  At
      OUT     M533  ; Conv'   #17 On  At
      MPP
      OUT     T24 K100  ; Conv'   #16->#17MoveOverTm
797   LDI     X56  ; Conv'   #17 StopPh
      ANI     T24  ; Conv'   #16->#17MoveOverTm
      MPS
      INV
      RST     L115  ; COnv    #16->#17Move    Latch
      MPP
      ANI     M1101  ; ConveyorTotal   Alarm
      AND     M101  ; Auto    Mode
      INV
      RST     M530  ; Conv    #16->#17Move Set
807   LD      M150  ; Auto    Start
      LD      X56  ; Conv'   #17 StopPh
      OR      L116  ; COnv    #17->#18Move    Latch
      ANB
      ANI     X57  ; Conv'   #18 StopPh
      ANI     M550  ; Conv    #18->#19Move Set
      SET     M540  ; Conv    #17->#18Move Set
      SET     L116  ; COnv    #17->#18Move    Latch
815   LD      M540  ; Conv    #17->#18Move Set
      MPS
      AND     SM400  ; Normal  On
      OUT     M542  ; Conv'   #17 On  At
      OUT     M543  ; Conv'   #18 On  At
      MPP
      OUT     T25 K100  ; Conv'   #17->#18MoveOverTm
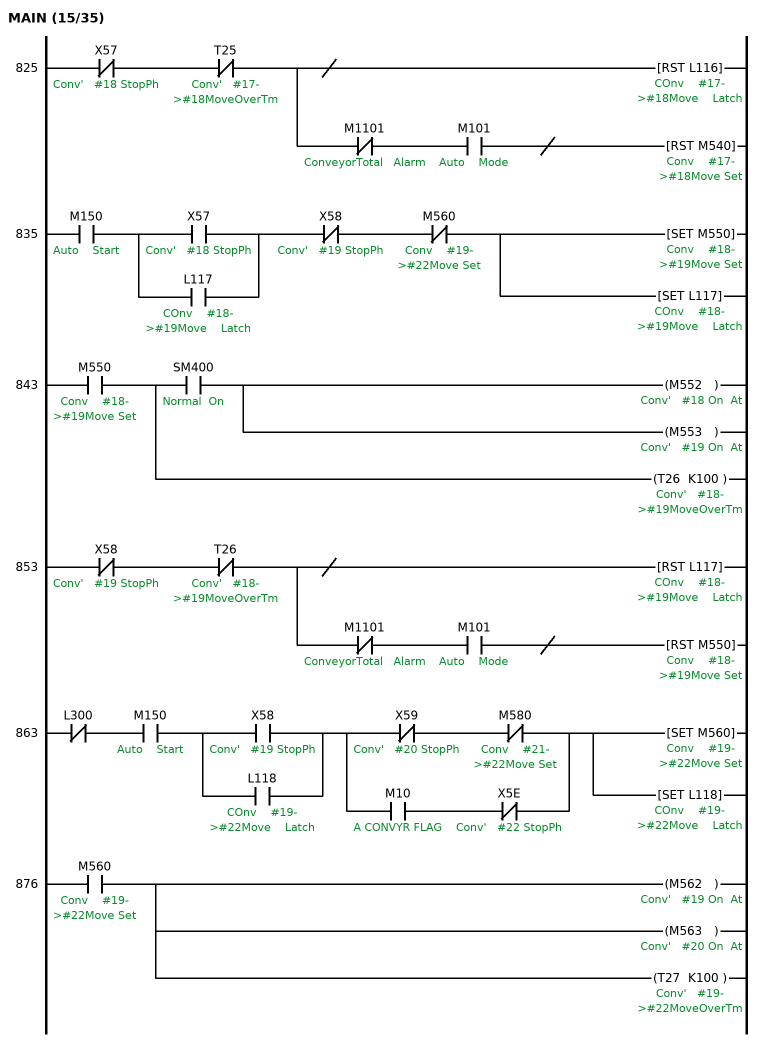
825   LDI     X57  ; Conv'   #18 StopPh
      ANI     T25  ; Conv'   #17->#18MoveOverTm
      MPS
      INV
      RST     L116  ; COnv    #17->#18Move    Latch
      MPP
      ANI     M1101  ; ConveyorTotal   Alarm
      AND     M101  ; Auto    Mode
      INV
      RST     M540  ; Conv    #17->#18Move Set
835   LD      M150  ; Auto    Start
      LD      X57  ; Conv'   #18 StopPh
      OR      L117  ; COnv    #18->#19Move    Latch
      ANB
      ANI     X58  ; Conv'   #19 StopPh
      ANI     M560  ; Conv    #19->#22Move Set
      SET     M550  ; Conv    #18->#19Move Set
      SET     L117  ; COnv    #18->#19Move    Latch
843   LD      M550  ; Conv    #18->#19Move Set
      MPS
      AND     SM400  ; Normal  On
      OUT     M552  ; Conv'   #18 On  At
      OUT     M553  ; Conv'   #19 On  At
      MPP
      OUT     T26 K100  ; Conv'   #18->#19MoveOverTm
853   LDI     X58  ; Conv'   #19 StopPh
      ANI     T26  ; Conv'   #18->#19MoveOverTm
      MPS
      INV
      RST     L117  ; COnv    #18->#19Move    Latch
      MPP
      ANI     M1101  ; ConveyorTotal   Alarm
      AND     M101  ; Auto    Mode
      INV
      RST     M550  ; Conv    #18->#19Move Set
863   LDI     L300
      AND     M150  ; Auto    Start
      LD      X58  ; Conv'   #19 StopPh
      OR      L118  ; COnv    #19->#22Move    Latch
      ANB
      LDI     X59  ; Conv'   #20 StopPh
      ANI     M580  ; Conv    #21->#22Move Set
      LD      M10  ; A CONVYR FLAG
      ANI     X5E  ; Conv'   #22 StopPh
      ORB
      ANB
      SET     M560  ; Conv    #19->#22Move Set
      SET     L118  ; COnv    #19->#22Move    Latch
876   LD      M560  ; Conv    #19->#22Move Set
      OUT     M562  ; Conv'   #19 On  At
      OUT     M563  ; Conv'   #20 On  At
      OUT     T27 K100  ; Conv'   #19->#22MoveOverTm
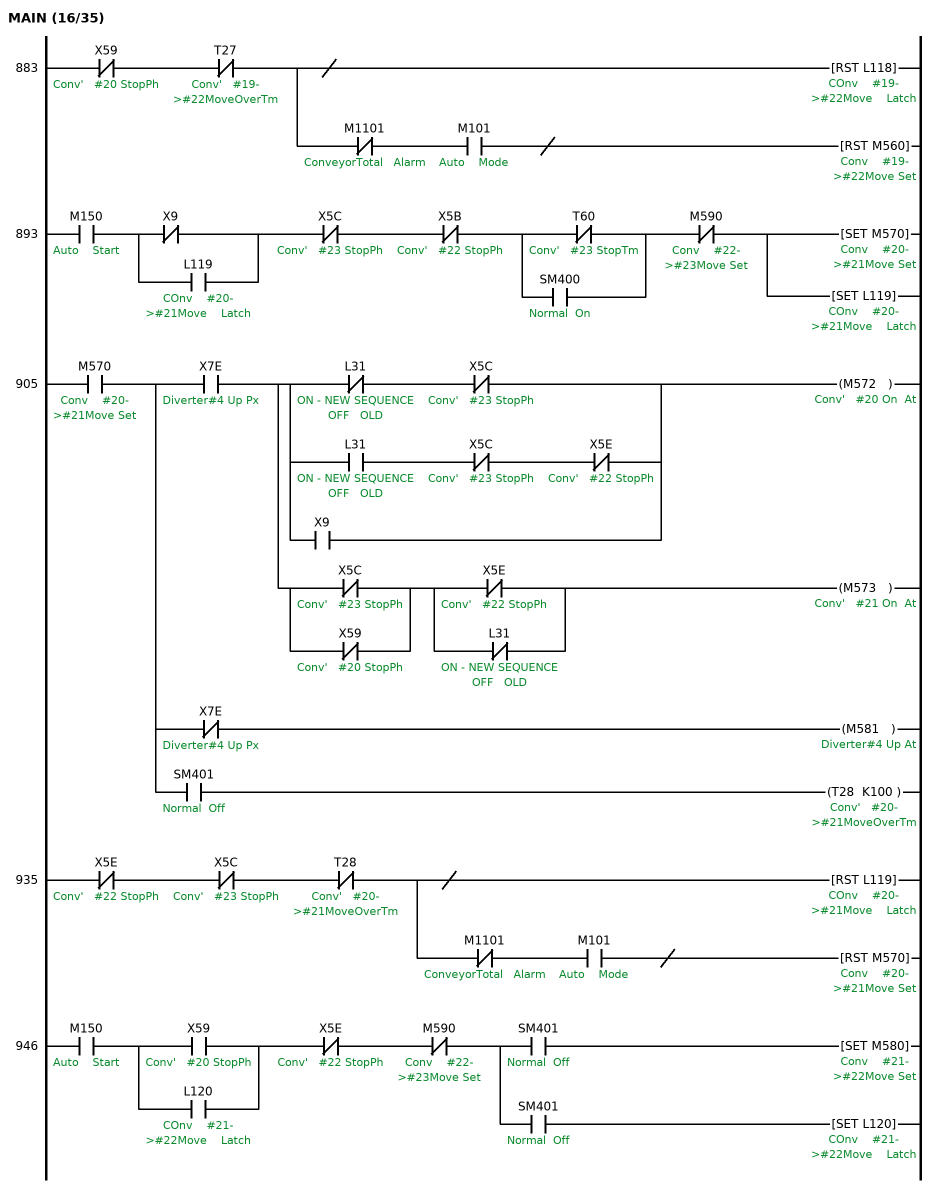
883   LDI     X59  ; Conv'   #20 StopPh
      ANI     T27  ; Conv'   #19->#22MoveOverTm
      MPS
      INV
      RST     L118  ; COnv    #19->#22Move    Latch
      MPP
      ANI     M1101  ; ConveyorTotal   Alarm
      AND     M101  ; Auto    Mode
      INV
      RST     M560  ; Conv    #19->#22Move Set
893   LD      M150  ; Auto    Start
      LDI     X9
      OR      L119  ; COnv    #20->#21Move    Latch
      ANB
      ANI     X5C  ; Conv'   #23 StopPh
      ANI     X5B  ; Conv'   #22 StopPh
      LDI     T60  ; Conv'   #23 StopTm
      OR      SM400  ; Normal  On
      ANB
      ANI     M590  ; Conv    #22->#23Move Set
      SET     M570  ; Conv    #20->#21Move Set
      SET     L119  ; COnv    #20->#21Move    Latch
905   LD      M570  ; Conv    #20->#21Move Set
      MPS
      AND     X7E  ; Diverter#4 Up Px
      MPS
      LDI     L31  ; ON - NEW SEQUENCE OFF   OLD
      ANI     X5C  ; Conv'   #23 StopPh
      LD      L31  ; ON - NEW SEQUENCE OFF   OLD
      ANI     X5C  ; Conv'   #23 StopPh
      ANI     X5E  ; Conv'   #22 StopPh
      ORB
      OR      X9
      ANB
      OUT     M572  ; Conv'   #20 On  At
      MPP
      LDI     X5C  ; Conv'   #23 StopPh
      ORI     X59  ; Conv'   #20 StopPh
      ANB
      LDI     X5E  ; Conv'   #22 StopPh
      ORI     L31  ; ON - NEW SEQUENCE OFF   OLD
      ANB
      OUT     M573  ; Conv'   #21 On  At
      MRD
      ANI     X7E  ; Diverter#4 Up Px
      OUT     M581  ; Diverter#4 Up At
      MPP
      AND     SM401  ; Normal  Off
      OUT     T28 K100  ; Conv'   #20->#21MoveOverTm
935   LDI     X5E  ; Conv'   #22 StopPh
      ANI     X5C  ; Conv'   #23 StopPh
      ANI     T28  ; Conv'   #20->#21MoveOverTm
      MPS
      INV
      RST     L119  ; COnv    #20->#21Move    Latch
      MPP
      ANI     M1101  ; ConveyorTotal   Alarm
      AND     M101  ; Auto    Mode
      INV
      RST     M570  ; Conv    #20->#21Move Set
946   LD      M150  ; Auto    Start
      LD      X59  ; Conv'   #20 StopPh
      OR      L120  ; COnv    #21->#22Move    Latch
      ANB
      ANI     X5E  ; Conv'   #22 StopPh
      ANI     M590  ; Conv    #22->#23Move Set
      MPS
      AND     SM401  ; Normal  Off
      SET     M580  ; Conv    #21->#22Move Set
      MPP
      AND     SM401  ; Normal  Off
      SET     L120  ; COnv    #21->#22Move    Latch
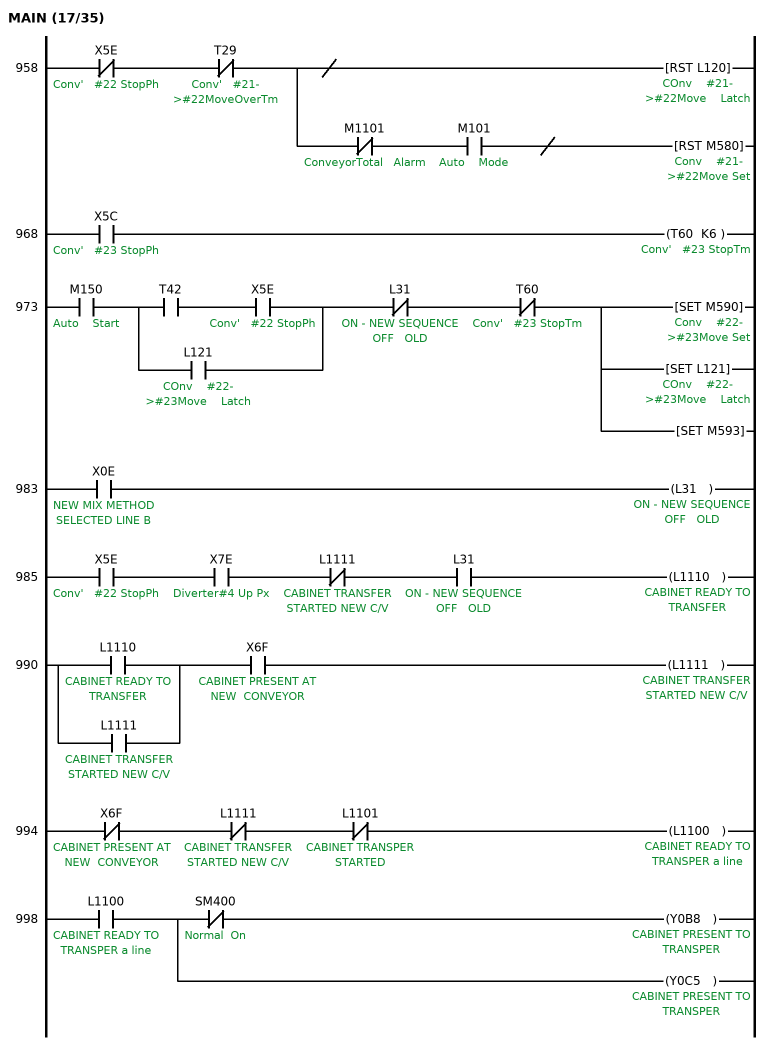
958   LDI     X5E  ; Conv'   #22 StopPh
      ANI     T29  ; Conv'   #21->#22MoveOverTm
      MPS
      INV
      RST     L120  ; COnv    #21->#22Move    Latch
      MPP
      ANI     M1101  ; ConveyorTotal   Alarm
      AND     M101  ; Auto    Mode
      INV
      RST     M580  ; Conv    #21->#22Move Set
968   LD      X5C  ; Conv'   #23 StopPh
      OUT     T60 K6  ; Conv'   #23 StopTm
973   LD      M150  ; Auto    Start
      LD      T42
      AND     X5E  ; Conv'   #22 StopPh
      OR      L121  ; COnv    #22->#23Move    Latch
      ANB
      ANI     L31  ; ON - NEW SEQUENCE OFF   OLD
      ANI     T60  ; Conv'   #23 StopTm
      SET     M590  ; Conv    #22->#23Move Set
      SET     L121  ; COnv    #22->#23Move    Latch
      SET     M593
983   LD      X0E  ; NEW MIX METHOD  SELECTED LINE B
      OUT     L31  ; ON - NEW SEQUENCE OFF   OLD
985   LD      X5E  ; Conv'   #22 StopPh
      AND     X7E  ; Diverter#4 Up Px
      ANI     L1111  ; CABINET TRANSFER STARTED NEW C/V
      AND     L31  ; ON - NEW SEQUENCE OFF   OLD
      OUT     L1110  ; CABINET READY TO TRANSFER
990   LD      L1110  ; CABINET READY TO TRANSFER
      OR      L1111  ; CABINET TRANSFER STARTED NEW C/V
      AND     X6F  ; CABINET PRESENT AT NEW  CONVEYOR
      OUT     L1111  ; CABINET TRANSFER STARTED NEW C/V
994   LDI     X6F  ; CABINET PRESENT AT NEW  CONVEYOR
      ANI     L1111  ; CABINET TRANSFER STARTED NEW C/V
      ANI     L1101  ; CABINET TRANSPER STARTED
      OUT     L1100  ; CABINET READY TO TRANSPER a line
998   LD      L1100  ; CABINET READY TO TRANSPER a line
      MPS
      ANI     SM400  ; Normal  On
      OUT     Y0B8  ; CABINET PRESENT TO      TRANSPER
      MPP
      OUT     Y0C5  ; CABINET PRESENT TO      TRANSPER
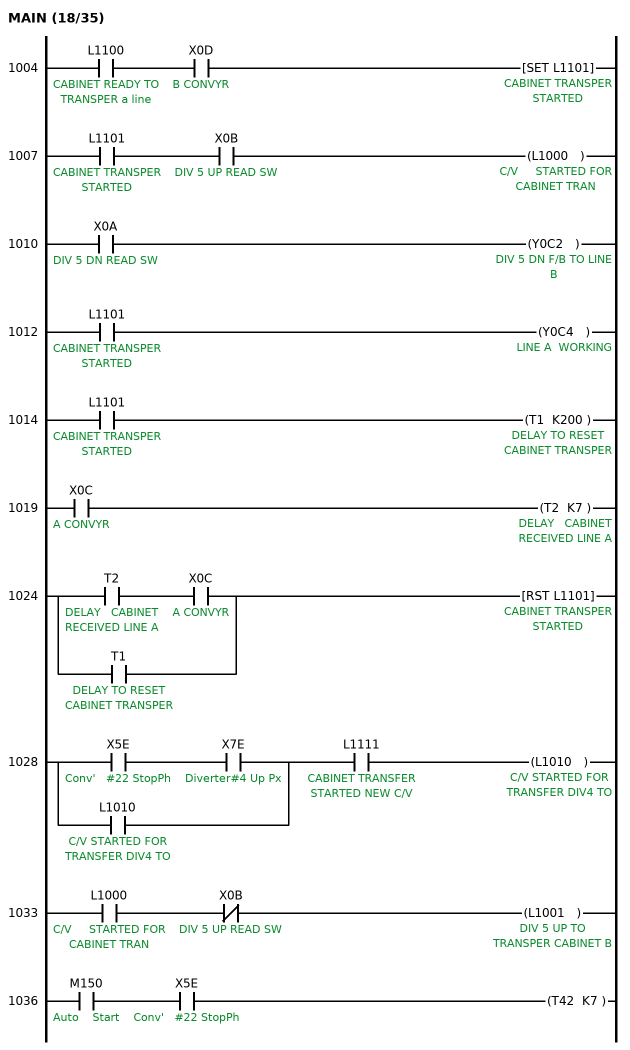
1004  LD      L1100  ; CABINET READY TO TRANSPER a line
      AND     X0D  ; B CONVYR
      SET     L1101  ; CABINET TRANSPER STARTED
1007  LD      L1101  ; CABINET TRANSPER STARTED
      AND     X0B  ; DIV 5 UP READ SW
      OUT     L1000  ; C/V     STARTED FOR CABINET TRAN
1010  LD      X0A  ; DIV 5 DN READ SW
      OUT     Y0C2  ; DIV 5 DN F/B TO LINE B
1012  LD      L1101  ; CABINET TRANSPER STARTED
      OUT     Y0C4  ; LINE A  WORKING
1014  LD      L1101  ; CABINET TRANSPER STARTED
      OUT     T1 K200  ; DELAY TO RESET CABINET TRANSPER
1019  LD      X0C  ; A CONVYR
      OUT     T2 K7  ; DELAY   CABINET RECEIVED LINE A
1024  LD      T2  ; DELAY   CABINET RECEIVED LINE A
      AND     X0C  ; A CONVYR
      OR      T1  ; DELAY TO RESET CABINET TRANSPER
      RST     L1101  ; CABINET TRANSPER STARTED
1028  LD      X5E  ; Conv'   #22 StopPh
      AND     X7E  ; Diverter#4 Up Px
      OR      L1010  ; C/V STARTED FOR TRANSFER DIV4 TO
      AND     L1111  ; CABINET TRANSFER STARTED NEW C/V
      OUT     L1010  ; C/V STARTED FOR TRANSFER DIV4 TO
1033  LD      L1000  ; C/V     STARTED FOR CABINET TRAN
      ANI     X0B  ; DIV 5 UP READ SW
      OUT     L1001  ; DIV 5 UP TO TRANSPER CABINET B
1036  LD      M150  ; Auto    Start
      AND     X5E  ; Conv'   #22 StopPh
      OUT     T42 K7
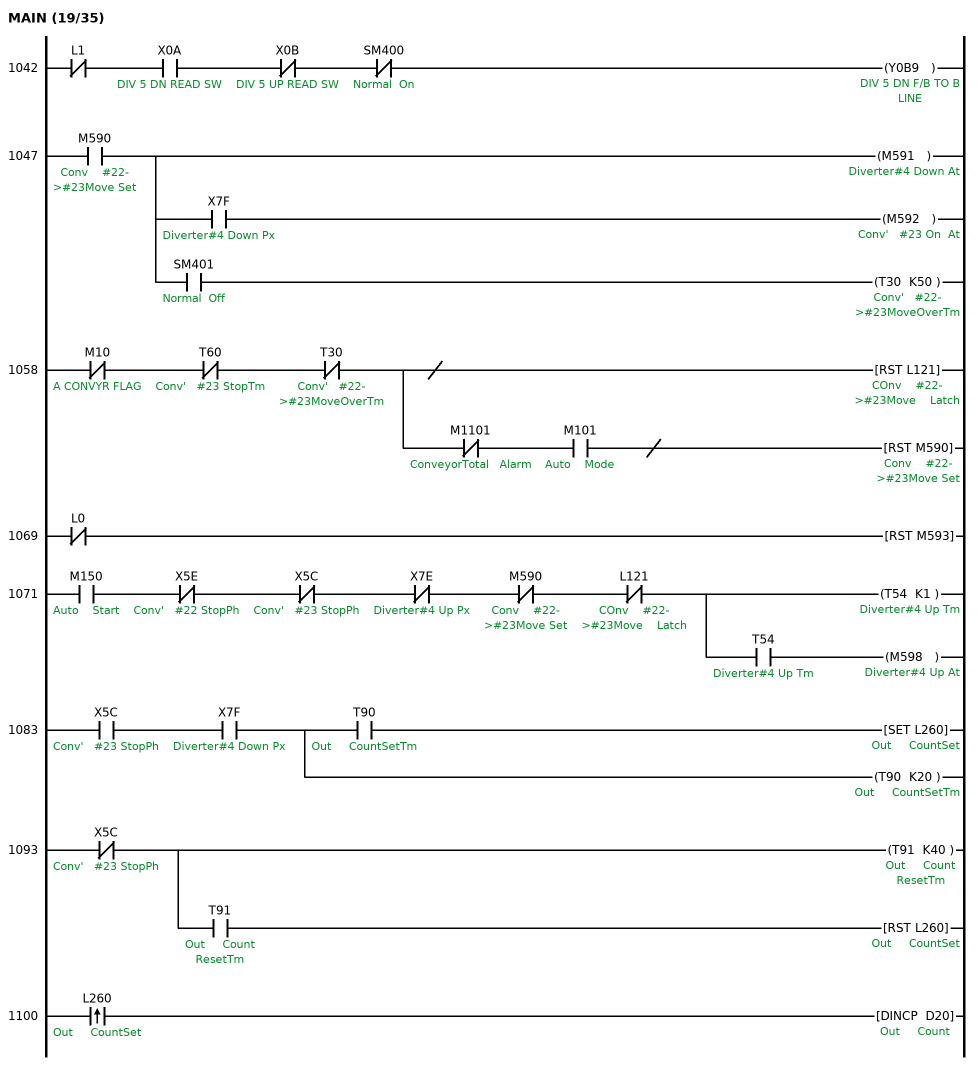
1042  LDI     L1
      AND     X0A  ; DIV 5 DN READ SW
      ANI     X0B  ; DIV 5 UP READ SW
      ANI     SM400  ; Normal  On
      OUT     Y0B9  ; DIV 5 DN F/B TO B LINE
1047  LD      M590  ; Conv    #22->#23Move Set
      OUT     M591  ; Diverter#4 Down At
      MPS
      AND     X7F  ; Diverter#4 Down Px
      OUT     M592  ; Conv'   #23 On  At
      MPP
      AND     SM401  ; Normal  Off
      OUT     T30 K50  ; Conv'   #22->#23MoveOverTm
1058  LDI     M10  ; A CONVYR FLAG
      ANI     T60  ; Conv'   #23 StopTm
      ANI     T30  ; Conv'   #22->#23MoveOverTm
      MPS
      INV
      RST     L121  ; COnv    #22->#23Move    Latch
      MPP
      ANI     M1101  ; ConveyorTotal   Alarm
      AND     M101  ; Auto    Mode
      INV
      RST     M590  ; Conv    #22->#23Move Set
1069  LDI     L0
      RST     M593
1071  LD      M150  ; Auto    Start
      ANI     X5E  ; Conv'   #22 StopPh
      ANI     X5C  ; Conv'   #23 StopPh
      ANI     X7E  ; Diverter#4 Up Px
      ANI     M590  ; Conv    #22->#23Move Set
      ANI     L121  ; COnv    #22->#23Move    Latch
      OUT     T54 K1  ; Diverter#4 Up Tm
      AND     T54  ; Diverter#4 Up Tm
      OUT     M598  ; Diverter#4 Up At
1083  LD      X5C  ; Conv'   #23 StopPh
      AND     X7F  ; Diverter#4 Down Px
      MPS
      AND     T90  ; Out     CountSetTm
      SET     L260  ; Out     CountSet
      MPP
      OUT     T90 K20  ; Out     CountSetTm
1093  LDI     X5C  ; Conv'   #23 StopPh
      OUT     T91 K40  ; Out     Count   ResetTm
      AND     T91  ; Out     Count   ResetTm
      RST     L260  ; Out     CountSet
1100  LDP     L260  ; Out     CountSet
      DINCP   D20  ; Out     Count
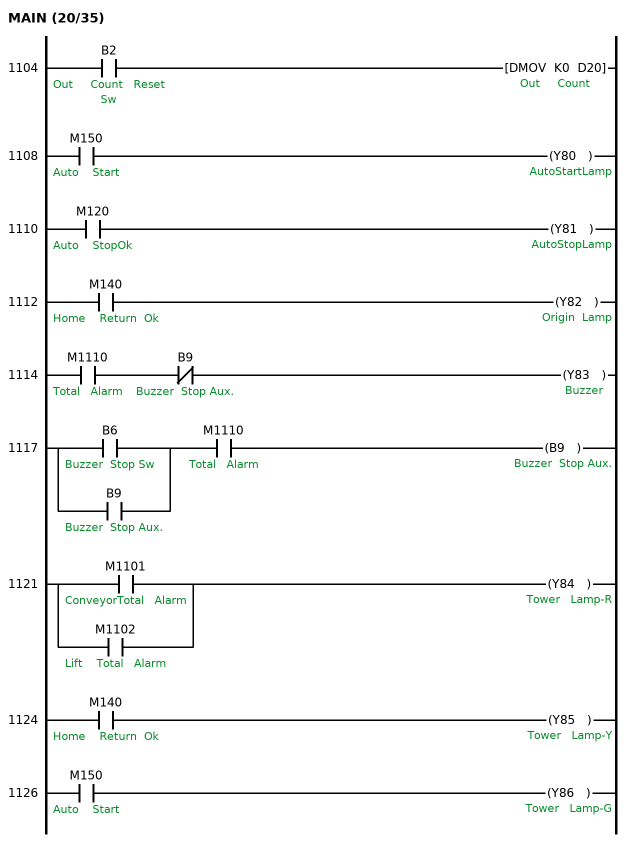
1104  LD      B2  ; Out     Count   Reset Sw
      DMOV    K0 D20
1108  LD      M150  ; Auto    Start
      OUT     Y80  ; AutoStartLamp
1110  LD      M120  ; Auto    StopOk
      OUT     Y81  ; AutoStopLamp
1112  LD      M140  ; Home    Return  Ok
      OUT     Y82  ; Origin  Lamp
1114  LD      M1110  ; Total   Alarm
      ANI     B9  ; Buzzer  Stop Aux.
      OUT     Y83  ; Buzzer
1117  LD      B6  ; Buzzer  Stop Sw
      OR      B9  ; Buzzer  Stop Aux.
      AND     M1110  ; Total   Alarm
      OUT     B9  ; Buzzer  Stop Aux.
1121  LD      M1101  ; ConveyorTotal   Alarm
      OR      M1102  ; Lift    Total   Alarm
      OUT     Y84  ; Tower   Lamp-R
1124  LD      M140  ; Home    Return  Ok
      OUT     Y85  ; Tower   Lamp-Y
1126  LD      M150  ; Auto    Start
      OUT     Y86  ; Tower   Lamp-G
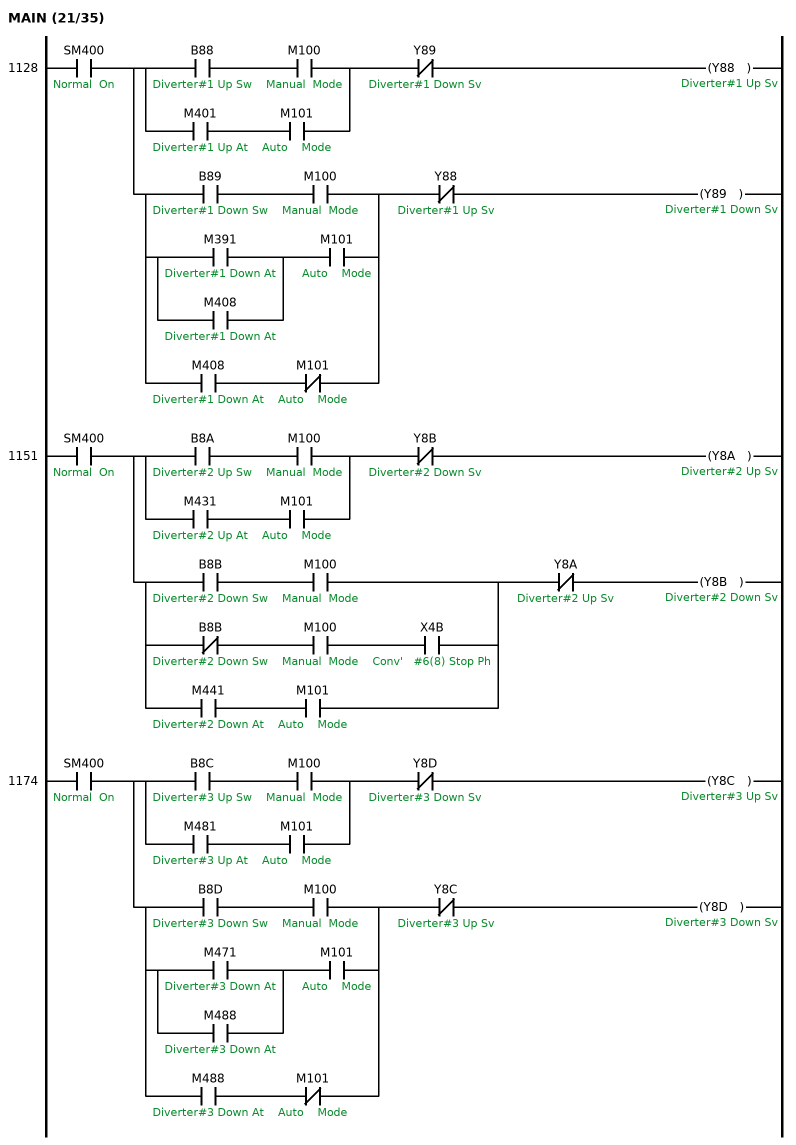
1128  LD      SM400  ; Normal  On
      MPS
      LD      B88  ; Diverter#1 Up Sw
      AND     M100  ; Manual  Mode
      LD      M401  ; Diverter#1 Up At
      AND     M101  ; Auto    Mode
      ORB
      ANB
      ANI     Y89  ; Diverter#1 Down Sv
      OUT     Y88  ; Diverter#1 Up Sv
      MPP
      LD      B89  ; Diverter#1 Down Sw
      AND     M100  ; Manual  Mode
      LD      M391  ; Diverter#1 Down At
      OR      M408  ; Diverter#1 Down At
      AND     M101  ; Auto    Mode
      ORB
      LD      M408  ; Diverter#1 Down At
      ANI     M101  ; Auto    Mode
      ORB
      ANB
      ANI     Y88  ; Diverter#1 Up Sv
      OUT     Y89  ; Diverter#1 Down Sv
1151  LD      SM400  ; Normal  On
      MPS
      LD      B8A  ; Diverter#2 Up Sw
      AND     M100  ; Manual  Mode
      LD      M431  ; Diverter#2 Up At
      AND     M101  ; Auto    Mode
      ORB
      ANB
      ANI     Y8B  ; Diverter#2 Down Sv
      OUT     Y8A  ; Diverter#2 Up Sv
      MPP
      LD      B8B  ; Diverter#2 Down Sw
      AND     M100  ; Manual  Mode
      LDI     B8B  ; Diverter#2 Down Sw
      AND     M100  ; Manual  Mode
      AND     X4B  ; Conv'   #6(8) Stop Ph
      ORB
      LD      M441  ; Diverter#2 Down At
      AND     M101  ; Auto    Mode
      ORB
      ANB
      ANI     Y8A  ; Diverter#2 Up Sv
      OUT     Y8B  ; Diverter#2 Down Sv
1174  LD      SM400  ; Normal  On
      MPS
      LD      B8C  ; Diverter#3 Up Sw
      AND     M100  ; Manual  Mode
      LD      M481  ; Diverter#3 Up At
      AND     M101  ; Auto    Mode
      ORB
      ANB
      ANI     Y8D  ; Diverter#3 Down Sv
      OUT     Y8C  ; Diverter#3 Up Sv
      MPP
      LD      B8D  ; Diverter#3 Down Sw
      AND     M100  ; Manual  Mode
      LD      M471  ; Diverter#3 Down At
      OR      M488  ; Diverter#3 Down At
      AND     M101  ; Auto    Mode
      ORB
      LD      M488  ; Diverter#3 Down At
      ANI     M101  ; Auto    Mode
      ORB
      ANB
      ANI     Y8C  ; Diverter#3 Up Sv
      OUT     Y8D  ; Diverter#3 Down Sv
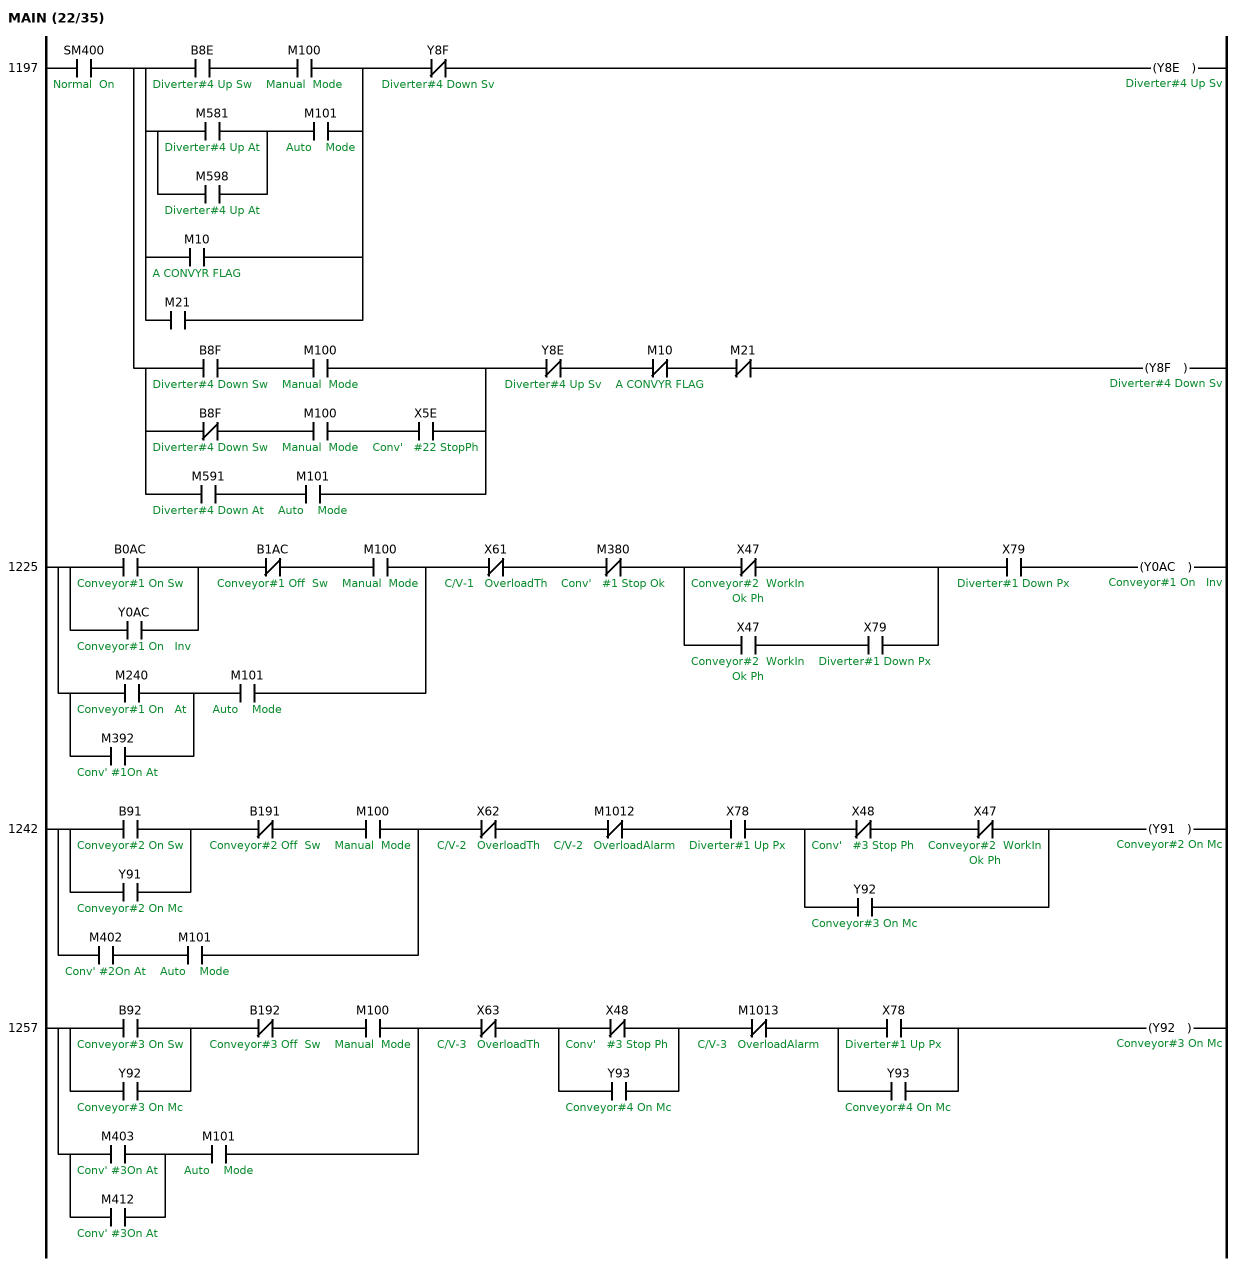
1197  LD      SM400  ; Normal  On
      MPS
      LD      B8E  ; Diverter#4 Up Sw
      AND     M100  ; Manual  Mode
      LD      M581  ; Diverter#4 Up At
      OR      M598  ; Diverter#4 Up At
      AND     M101  ; Auto    Mode
      ORB
      OR      M10  ; A CONVYR FLAG
      OR      M21
      ANB
      ANI     Y8F  ; Diverter#4 Down Sv
      OUT     Y8E  ; Diverter#4 Up Sv
      MPP
      LD      B8F  ; Diverter#4 Down Sw
      AND     M100  ; Manual  Mode
      LDI     B8F  ; Diverter#4 Down Sw
      AND     M100  ; Manual  Mode
      AND     X5E  ; Conv'   #22 StopPh
      ORB
      LD      M591  ; Diverter#4 Down At
      AND     M101  ; Auto    Mode
      ORB
      ANB
      ANI     Y8E  ; Diverter#4 Up Sv
      ANI     M10  ; A CONVYR FLAG
      ANI     M21
      OUT     Y8F  ; Diverter#4 Down Sv
1225  LD      B0AC  ; Conveyor#1 On Sw
      OR      Y0AC  ; Conveyor#1 On   Inv
      ANI     B1AC  ; Conveyor#1 Off  Sw
      AND     M100  ; Manual  Mode
      LD      M240  ; Conveyor#1 On   At
      OR      M392  ; Conv' #1On At
      AND     M101  ; Auto    Mode
      ORB
      ANI     X61  ; C/V-1   OverloadTh
      ANI     M380  ; Conv'   #1 Stop Ok
      LDI     X47  ; Conveyor#2  WorkIn Ok Ph
      LD      X47  ; Conveyor#2  WorkIn Ok Ph
      AND     X79  ; Diverter#1 Down Px
      ORB
      ANB
      AND     X79  ; Diverter#1 Down Px
      OUT     Y0AC  ; Conveyor#1 On   Inv
1242  LD      B91  ; Conveyor#2 On Sw
      OR      Y91  ; Conveyor#2 On Mc
      ANI     B191  ; Conveyor#2 Off  Sw
      AND     M100  ; Manual  Mode
      LD      M402  ; Conv' #2On At
      AND     M101  ; Auto    Mode
      ORB
      ANI     X62  ; C/V-2   OverloadTh
      ANI     M1012  ; C/V-2   OverloadAlarm
      AND     X78  ; Diverter#1 Up Px
      LDI     X48  ; Conv'   #3 Stop Ph
      ANI     X47  ; Conveyor#2  WorkIn Ok Ph
      OR      Y92  ; Conveyor#3 On Mc
      ANB
      OUT     Y91  ; Conveyor#2 On Mc
1257  LD      B92  ; Conveyor#3 On Sw
      OR      Y92  ; Conveyor#3 On Mc
      ANI     B192  ; Conveyor#3 Off  Sw
      AND     M100  ; Manual  Mode
      LD      M403  ; Conv' #3On At
      OR      M412  ; Conv' #3On At
      AND     M101  ; Auto    Mode
      ORB
      ANI     X63  ; C/V-3   OverloadTh
      LDI     X48  ; Conv'   #3 Stop Ph
      OR      Y93  ; Conveyor#4 On Mc
      ANB
      ANI     M1013  ; C/V-3   OverloadAlarm
      LD      X78  ; Diverter#1 Up Px
      OR      Y93  ; Conveyor#4 On Mc
      ANB
      OUT     Y92  ; Conveyor#3 On Mc
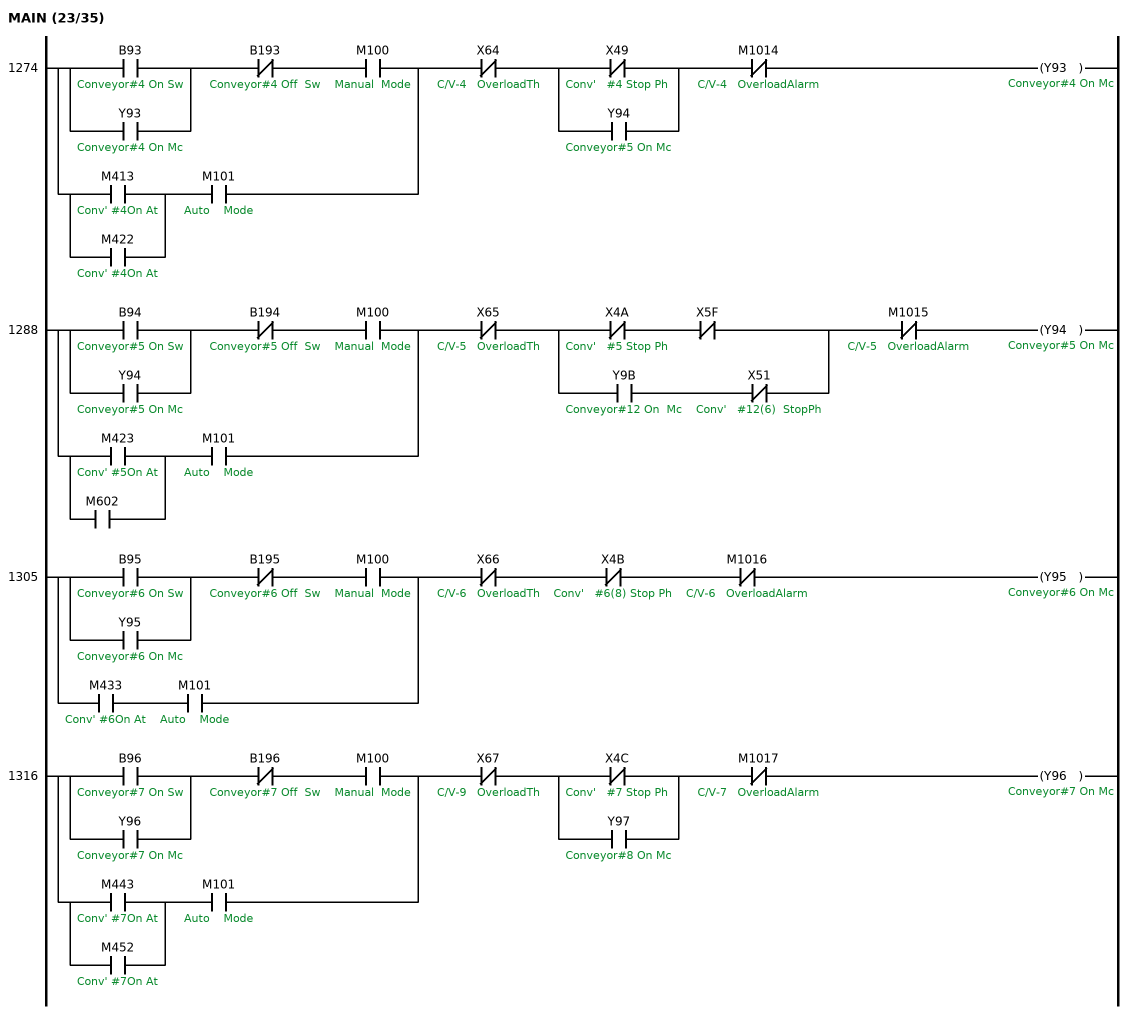
1274  LD      B93  ; Conveyor#4 On Sw
      OR      Y93  ; Conveyor#4 On Mc
      ANI     B193  ; Conveyor#4 Off  Sw
      AND     M100  ; Manual  Mode
      LD      M413  ; Conv' #4On At
      OR      M422  ; Conv' #4On At
      AND     M101  ; Auto    Mode
      ORB
      ANI     X64  ; C/V-4   OverloadTh
      LDI     X49  ; Conv'   #4 Stop Ph
      OR      Y94  ; Conveyor#5 On Mc
      ANB
      ANI     M1014  ; C/V-4   OverloadAlarm
      OUT     Y93  ; Conveyor#4 On Mc
1288  LD      B94  ; Conveyor#5 On Sw
      OR      Y94  ; Conveyor#5 On Mc
      ANI     B194  ; Conveyor#5 Off  Sw
      AND     M100  ; Manual  Mode
      LD      M423  ; Conv' #5On At
      OR      M602
      AND     M101  ; Auto    Mode
      ORB
      ANI     X65  ; C/V-5   OverloadTh
      LDI     X4A  ; Conv'   #5 Stop Ph
      ANI     X5F
      LD      Y9B  ; Conveyor#12 On  Mc
      ANI     X51  ; Conv'   #12(6)  StopPh
      ORB
      ANB
      ANI     M1015  ; C/V-5   OverloadAlarm
      OUT     Y94  ; Conveyor#5 On Mc
1305  LD      B95  ; Conveyor#6 On Sw
      OR      Y95  ; Conveyor#6 On Mc
      ANI     B195  ; Conveyor#6 Off  Sw
      AND     M100  ; Manual  Mode
      LD      M433  ; Conv' #6On At
      AND     M101  ; Auto    Mode
      ORB
      ANI     X66  ; C/V-6   OverloadTh
      ANI     X4B  ; Conv'   #6(8) Stop Ph
      ANI     M1016  ; C/V-6   OverloadAlarm
      OUT     Y95  ; Conveyor#6 On Mc
1316  LD      B96  ; Conveyor#7 On Sw
      OR      Y96  ; Conveyor#7 On Mc
      ANI     B196  ; Conveyor#7 Off  Sw
      AND     M100  ; Manual  Mode
      LD      M443  ; Conv' #7On At
      OR      M452  ; Conv' #7On At
      AND     M101  ; Auto    Mode
      ORB
      ANI     X67  ; C/V-9   OverloadTh
      LDI     X4C  ; Conv'   #7 Stop Ph
      OR      Y97  ; Conveyor#8 On Mc
      ANB
      ANI     M1017  ; C/V-7   OverloadAlarm
      OUT     Y96  ; Conveyor#7 On Mc
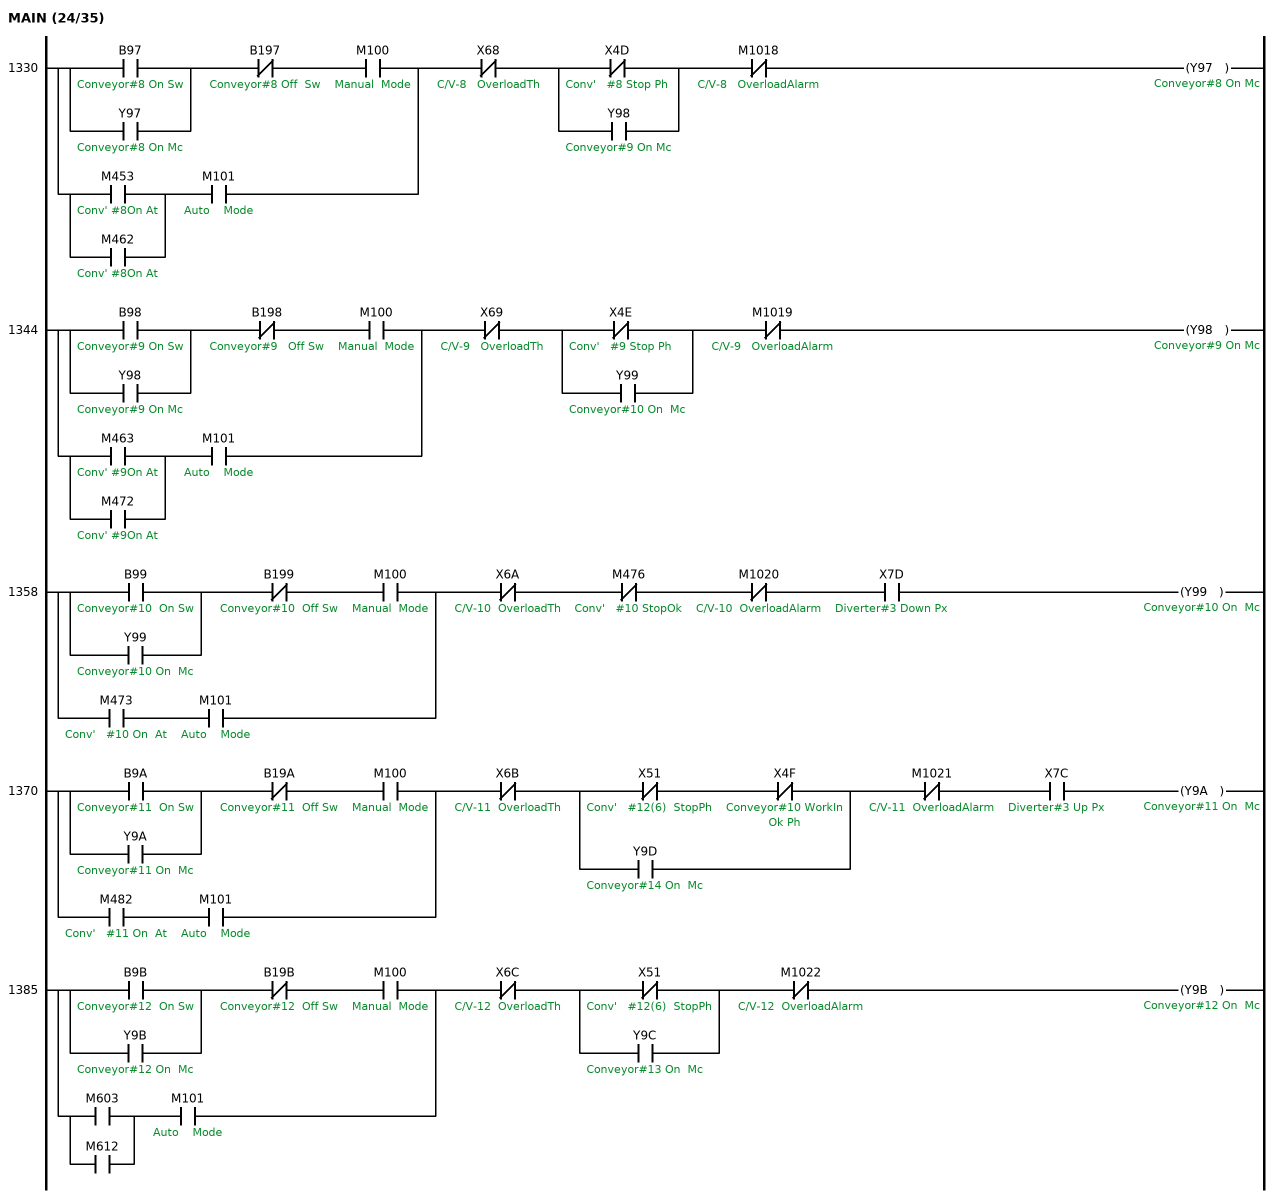
1330  LD      B97  ; Conveyor#8 On Sw
      OR      Y97  ; Conveyor#8 On Mc
      ANI     B197  ; Conveyor#8 Off  Sw
      AND     M100  ; Manual  Mode
      LD      M453  ; Conv' #8On At
      OR      M462  ; Conv' #8On At
      AND     M101  ; Auto    Mode
      ORB
      ANI     X68  ; C/V-8   OverloadTh
      LDI     X4D  ; Conv'   #8 Stop Ph
      OR      Y98  ; Conveyor#9 On Mc
      ANB
      ANI     M1018  ; C/V-8   OverloadAlarm
      OUT     Y97  ; Conveyor#8 On Mc
1344  LD      B98  ; Conveyor#9 On Sw
      OR      Y98  ; Conveyor#9 On Mc
      ANI     B198  ; Conveyor#9   Off Sw
      AND     M100  ; Manual  Mode
      LD      M463  ; Conv' #9On At
      OR      M472  ; Conv' #9On At
      AND     M101  ; Auto    Mode
      ORB
      ANI     X69  ; C/V-9   OverloadTh
      LDI     X4E  ; Conv'   #9 Stop Ph
      OR      Y99  ; Conveyor#10 On  Mc
      ANB
      ANI     M1019  ; C/V-9   OverloadAlarm
      OUT     Y98  ; Conveyor#9 On Mc
1358  LD      B99  ; Conveyor#10  On Sw
      OR      Y99  ; Conveyor#10 On  Mc
      ANI     B199  ; Conveyor#10  Off Sw
      AND     M100  ; Manual  Mode
      LD      M473  ; Conv'   #10 On  At
      AND     M101  ; Auto    Mode
      ORB
      ANI     X6A  ; C/V-10  OverloadTh
      ANI     M476  ; Conv'   #10 StopOk
      ANI     M1020  ; C/V-10  OverloadAlarm
      AND     X7D  ; Diverter#3 Down Px
      OUT     Y99  ; Conveyor#10 On  Mc
1370  LD      B9A  ; Conveyor#11  On Sw
      OR      Y9A  ; Conveyor#11 On  Mc
      ANI     B19A  ; Conveyor#11  Off Sw
      AND     M100  ; Manual  Mode
      LD      M482  ; Conv'   #11 On  At
      AND     M101  ; Auto    Mode
      ORB
      ANI     X6B  ; C/V-11  OverloadTh
      LDI     X51  ; Conv'   #12(6)  StopPh
      ANI     X4F  ; Conveyor#10 WorkIn Ok Ph
      OR      Y9D  ; Conveyor#14 On  Mc
      ANB
      ANI     M1021  ; C/V-11  OverloadAlarm
      AND     X7C  ; Diverter#3 Up Px
      OUT     Y9A  ; Conveyor#11 On  Mc
1385  LD      B9B  ; Conveyor#12  On Sw
      OR      Y9B  ; Conveyor#12 On  Mc
      ANI     B19B  ; Conveyor#12  Off Sw
      AND     M100  ; Manual  Mode
      LD      M603
      OR      M612
      AND     M101  ; Auto    Mode
      ORB
      ANI     X6C  ; C/V-12  OverloadTh
      LDI     X51  ; Conv'   #12(6)  StopPh
      OR      Y9C  ; Conveyor#13 On  Mc
      ANB
      ANI     M1022  ; C/V-12  OverloadAlarm
      OUT     Y9B  ; Conveyor#12 On  Mc
